//FloorStats 23
IF 
FB_BACnet_DAIKIN_MasterStation_III_No_6.StartStopStatus_064.bPresVal AND
FB_BACnet_DAIKIN_MasterStation_III_No_6.StartStopStatus_065.bPresVal AND
FB_BACnet_DAIKIN_MasterStation_III_No_6.StartStopStatus_066.bPresVal AND
FB_BACnet_DAIKIN_MasterStation_III_No_6.StartStopStatus_067.bPresVal AND
FB_BACnet_DAIKIN_MasterStation_III_No_6.StartStopStatus_068.bPresVal AND
FB_BACnet_DAIKIN_MasterStation_III_No_6.StartStopStatus_069.bPresVal AND
FB_BACnet_DAIKIN_MasterStation_III_No_6.StartStopStatus_070.bPresVal AND
FB_BACnet_DAIKIN_MasterStation_III_No_6.StartStopStatus_071.bPresVal AND
FB_BACnet_DAIKIN_MasterStation_III_No_6.StartStopStatus_072.bPresVal AND
FB_BACnet_DAIKIN_MasterStation_III_No_6.StartStopStatus_073.bPresVal AND
FB_BACnet_DAIKIN_MasterStation_III_No_6.StartStopStatus_074.bPresVal AND
FB_BACnet_DAIKIN_MasterStation_III_No_6.StartStopStatus_075.bPresVal AND
FB_BACnet_DAIKIN_MasterStation_III_No_6.StartStopStatus_076.bPresVal AND
FB_BACnet_DAIKIN_MasterStation_III_No_6.StartStopStatus_077.bPresVal AND
FB_BACnet_DAIKIN_MasterStation_III_No_6.StartStopStatus_078.bPresVal AND
FB_BACnet_DAIKIN_MasterStation_III_No_6.StartStopStatus_079.bPresVal AND
FB_BACnet_DAIKIN_MasterStation_III_No_6.StartStopStatus_080.bPresVal AND
FB_BACnet_DAIKIN_MasterStation_III_No_6.StartStopStatus_081.bPresVal AND
FB_BACnet_DAIKIN_MasterStation_III_No_6.StartStopStatus_082.bPresVal AND
FB_BACnet_DAIKIN_MasterStation_III_No_6.StartStopStatus_083.bPresVal AND
FB_BACnet_DAIKIN_MasterStation_III_No_6.StartStopStatus_224.bPresVal
THEN
	nFloorStatus23 := 1;
ELSIF
NOT FB_BACnet_DAIKIN_MasterStation_III_No_6.StartStopStatus_064.bPresVal AND
NOT FB_BACnet_DAIKIN_MasterStation_III_No_6.StartStopStatus_065.bPresVal AND
NOT FB_BACnet_DAIKIN_MasterStation_III_No_6.StartStopStatus_066.bPresVal AND
NOT FB_BACnet_DAIKIN_MasterStation_III_No_6.StartStopStatus_067.bPresVal AND
NOT FB_BACnet_DAIKIN_MasterStation_III_No_6.StartStopStatus_068.bPresVal AND
NOT FB_BACnet_DAIKIN_MasterStation_III_No_6.StartStopStatus_069.bPresVal AND
NOT FB_BACnet_DAIKIN_MasterStation_III_No_6.StartStopStatus_070.bPresVal AND
NOT FB_BACnet_DAIKIN_MasterStation_III_No_6.StartStopStatus_071.bPresVal AND
NOT FB_BACnet_DAIKIN_MasterStation_III_No_6.StartStopStatus_072.bPresVal AND
NOT FB_BACnet_DAIKIN_MasterStation_III_No_6.StartStopStatus_073.bPresVal AND
NOT FB_BACnet_DAIKIN_MasterStation_III_No_6.StartStopStatus_074.bPresVal AND
NOT FB_BACnet_DAIKIN_MasterStation_III_No_6.StartStopStatus_075.bPresVal AND
NOT FB_BACnet_DAIKIN_MasterStation_III_No_6.StartStopStatus_076.bPresVal AND
NOT FB_BACnet_DAIKIN_MasterStation_III_No_6.StartStopStatus_077.bPresVal AND
NOT FB_BACnet_DAIKIN_MasterStation_III_No_6.StartStopStatus_078.bPresVal AND
NOT FB_BACnet_DAIKIN_MasterStation_III_No_6.StartStopStatus_079.bPresVal AND
NOT FB_BACnet_DAIKIN_MasterStation_III_No_6.StartStopStatus_080.bPresVal AND
NOT FB_BACnet_DAIKIN_MasterStation_III_No_6.StartStopStatus_081.bPresVal AND
NOT FB_BACnet_DAIKIN_MasterStation_III_No_6.StartStopStatus_082.bPresVal AND
NOT FB_BACnet_DAIKIN_MasterStation_III_No_6.StartStopStatus_083.bPresVal AND
NOT FB_BACnet_DAIKIN_MasterStation_III_No_6.StartStopStatus_224.bPresVal
THEN
	nFloorStatus23 := 0;
ELSE
	nFloorStatus23 := 2;
END_IF

//FloorStats 25
IF 
FB_BACnet_DAIKIN_MasterStation_III_No_6.StartStopStatus_128.bPresVal AND
FB_BACnet_DAIKIN_MasterStation_III_No_6.StartStopStatus_129.bPresVal AND
FB_BACnet_DAIKIN_MasterStation_III_No_6.StartStopStatus_130.bPresVal AND
FB_BACnet_DAIKIN_MasterStation_III_No_6.StartStopStatus_131.bPresVal AND
FB_BACnet_DAIKIN_MasterStation_III_No_6.StartStopStatus_132.bPresVal AND
FB_BACnet_DAIKIN_MasterStation_III_No_6.StartStopStatus_133.bPresVal AND
//FB_BACnet_DAIKIN_MasterStation_III_No_6.StartStopStatus_134.bPresVal AND
//FB_BACnet_DAIKIN_MasterStation_III_No_6.StartStopStatus_135.bPresVal AND
FB_BACnet_DAIKIN_MasterStation_III_No_6.StartStopStatus_136.bPresVal AND
FB_BACnet_DAIKIN_MasterStation_III_No_6.StartStopStatus_137.bPresVal AND
FB_BACnet_DAIKIN_MasterStation_III_No_6.StartStopStatus_138.bPresVal AND
FB_BACnet_DAIKIN_MasterStation_III_No_6.StartStopStatus_139.bPresVal AND
FB_BACnet_DAIKIN_MasterStation_III_No_6.StartStopStatus_140.bPresVal AND
FB_BACnet_DAIKIN_MasterStation_III_No_6.StartStopStatus_141.bPresVal AND
FB_BACnet_DAIKIN_MasterStation_III_No_6.StartStopStatus_142.bPresVal AND
FB_BACnet_DAIKIN_MasterStation_III_No_6.StartStopStatus_143.bPresVal AND
FB_BACnet_DAIKIN_MasterStation_III_No_6.StartStopStatus_144.bPresVal AND
FB_BACnet_DAIKIN_MasterStation_III_No_6.StartStopStatus_145.bPresVal AND
FB_BACnet_DAIKIN_MasterStation_III_No_6.StartStopStatus_146.bPresVal AND
FB_BACnet_DAIKIN_MasterStation_III_No_6.StartStopStatus_147.bPresVal AND
FB_BACnet_DAIKIN_MasterStation_III_No_6.StartStopStatus_225.bPresVal AND
FB_BACnet_DAIKIN_MasterStation_III_No_6.StartStopStatus_241.bPresVal AND
FB_BACnet_DAIKIN_MasterStation_III_No_6.StartStopStatus_176.bPresVal
THEN
	nFloorStatus25 := 1;
ELSIF
NOT FB_BACnet_DAIKIN_MasterStation_III_No_6.StartStopStatus_128.bPresVal AND
NOT FB_BACnet_DAIKIN_MasterStation_III_No_6.StartStopStatus_129.bPresVal AND
NOT FB_BACnet_DAIKIN_MasterStation_III_No_6.StartStopStatus_130.bPresVal AND
NOT FB_BACnet_DAIKIN_MasterStation_III_No_6.StartStopStatus_131.bPresVal AND
NOT FB_BACnet_DAIKIN_MasterStation_III_No_6.StartStopStatus_132.bPresVal AND
NOT FB_BACnet_DAIKIN_MasterStation_III_No_6.StartStopStatus_133.bPresVal AND
//NOT FB_BACnet_DAIKIN_MasterStation_III_No_6.StartStopStatus_134.bPresVal AND
//NOT FB_BACnet_DAIKIN_MasterStation_III_No_6.StartStopStatus_135.bPresVal AND
NOT FB_BACnet_DAIKIN_MasterStation_III_No_6.StartStopStatus_136.bPresVal AND
NOT FB_BACnet_DAIKIN_MasterStation_III_No_6.StartStopStatus_137.bPresVal AND
NOT FB_BACnet_DAIKIN_MasterStation_III_No_6.StartStopStatus_138.bPresVal AND
NOT FB_BACnet_DAIKIN_MasterStation_III_No_6.StartStopStatus_139.bPresVal AND
NOT FB_BACnet_DAIKIN_MasterStation_III_No_6.StartStopStatus_140.bPresVal AND
NOT FB_BACnet_DAIKIN_MasterStation_III_No_6.StartStopStatus_141.bPresVal AND
NOT FB_BACnet_DAIKIN_MasterStation_III_No_6.StartStopStatus_142.bPresVal AND
NOT FB_BACnet_DAIKIN_MasterStation_III_No_6.StartStopStatus_143.bPresVal AND
NOT FB_BACnet_DAIKIN_MasterStation_III_No_6.StartStopStatus_144.bPresVal AND
NOT FB_BACnet_DAIKIN_MasterStation_III_No_6.StartStopStatus_145.bPresVal AND
NOT FB_BACnet_DAIKIN_MasterStation_III_No_6.StartStopStatus_146.bPresVal AND
NOT FB_BACnet_DAIKIN_MasterStation_III_No_6.StartStopStatus_147.bPresVal AND
NOT FB_BACnet_DAIKIN_MasterStation_III_No_6.StartStopStatus_225.bPresVal AND
NOT FB_BACnet_DAIKIN_MasterStation_III_No_6.StartStopStatus_241.bPresVal AND
NOT FB_BACnet_DAIKIN_MasterStation_III_No_6.StartStopStatus_176.bPresVal
THEN
	nFloorStatus25 := 0;
ELSE
	nFloorStatus25 := 2;
END_IF

//FloorStats 26
IF 
FB_BACnet_DAIKIN_MasterStation_III_No_6.StartStopStatus_192.bPresVal AND
FB_BACnet_DAIKIN_MasterStation_III_No_6.StartStopStatus_193.bPresVal AND
FB_BACnet_DAIKIN_MasterStation_III_No_6.StartStopStatus_194.bPresVal AND
FB_BACnet_DAIKIN_MasterStation_III_No_6.StartStopStatus_195.bPresVal AND
FB_BACnet_DAIKIN_MasterStation_III_No_6.StartStopStatus_196.bPresVal AND
FB_BACnet_DAIKIN_MasterStation_III_No_6.StartStopStatus_197.bPresVal AND
FB_BACnet_DAIKIN_MasterStation_III_No_6.StartStopStatus_198.bPresVal AND
FB_BACnet_DAIKIN_MasterStation_III_No_6.StartStopStatus_199.bPresVal AND
FB_BACnet_DAIKIN_MasterStation_III_No_6.StartStopStatus_200.bPresVal AND
FB_BACnet_DAIKIN_MasterStation_III_No_6.StartStopStatus_201.bPresVal AND
FB_BACnet_DAIKIN_MasterStation_III_No_6.StartStopStatus_202.bPresVal AND
FB_BACnet_DAIKIN_MasterStation_III_No_6.StartStopStatus_203.bPresVal AND
FB_BACnet_DAIKIN_MasterStation_III_No_6.StartStopStatus_204.bPresVal AND
FB_BACnet_DAIKIN_MasterStation_III_No_6.StartStopStatus_205.bPresVal AND
FB_BACnet_DAIKIN_MasterStation_III_No_6.StartStopStatus_206.bPresVal AND
FB_BACnet_DAIKIN_MasterStation_III_No_6.StartStopStatus_207.bPresVal AND
FB_BACnet_DAIKIN_MasterStation_III_No_6.StartStopStatus_208.bPresVal AND
FB_BACnet_DAIKIN_MasterStation_III_No_6.StartStopStatus_209.bPresVal AND
FB_BACnet_DAIKIN_MasterStation_III_No_6.StartStopStatus_210.bPresVal AND
FB_BACnet_DAIKIN_MasterStation_III_No_6.StartStopStatus_211.bPresVal AND
FB_BACnet_DAIKIN_MasterStation_III_No_6.StartStopStatus_226.bPresVal
THEN
	nFloorStatus26 := 1;
ELSIF
NOT FB_BACnet_DAIKIN_MasterStation_III_No_6.StartStopStatus_192.bPresVal AND
NOT FB_BACnet_DAIKIN_MasterStation_III_No_6.StartStopStatus_193.bPresVal AND
NOT FB_BACnet_DAIKIN_MasterStation_III_No_6.StartStopStatus_194.bPresVal AND
NOT FB_BACnet_DAIKIN_MasterStation_III_No_6.StartStopStatus_195.bPresVal AND
NOT FB_BACnet_DAIKIN_MasterStation_III_No_6.StartStopStatus_196.bPresVal AND
NOT FB_BACnet_DAIKIN_MasterStation_III_No_6.StartStopStatus_197.bPresVal AND
NOT FB_BACnet_DAIKIN_MasterStation_III_No_6.StartStopStatus_198.bPresVal AND
NOT FB_BACnet_DAIKIN_MasterStation_III_No_6.StartStopStatus_199.bPresVal AND
NOT FB_BACnet_DAIKIN_MasterStation_III_No_6.StartStopStatus_200.bPresVal AND
NOT FB_BACnet_DAIKIN_MasterStation_III_No_6.StartStopStatus_201.bPresVal AND
NOT FB_BACnet_DAIKIN_MasterStation_III_No_6.StartStopStatus_202.bPresVal AND
NOT FB_BACnet_DAIKIN_MasterStation_III_No_6.StartStopStatus_203.bPresVal AND
NOT FB_BACnet_DAIKIN_MasterStation_III_No_6.StartStopStatus_204.bPresVal AND
NOT FB_BACnet_DAIKIN_MasterStation_III_No_6.StartStopStatus_205.bPresVal AND
NOT FB_BACnet_DAIKIN_MasterStation_III_No_6.StartStopStatus_206.bPresVal AND
NOT FB_BACnet_DAIKIN_MasterStation_III_No_6.StartStopStatus_207.bPresVal AND
NOT FB_BACnet_DAIKIN_MasterStation_III_No_6.StartStopStatus_208.bPresVal AND
NOT FB_BACnet_DAIKIN_MasterStation_III_No_6.StartStopStatus_209.bPresVal AND
NOT FB_BACnet_DAIKIN_MasterStation_III_No_6.StartStopStatus_210.bPresVal AND
NOT FB_BACnet_DAIKIN_MasterStation_III_No_6.StartStopStatus_211.bPresVal AND
NOT FB_BACnet_DAIKIN_MasterStation_III_No_6.StartStopStatus_226.bPresVal
THEN
	nFloorStatus26 := 0;
ELSE
	nFloorStatus26 := 2;
END_IF

//FloorStats 27
IF 
FB_BACnet_DAIKIN_MasterStation_III_No_7.StartStopStatus_000.bPresVal AND
FB_BACnet_DAIKIN_MasterStation_III_No_7.StartStopStatus_001.bPresVal AND
FB_BACnet_DAIKIN_MasterStation_III_No_7.StartStopStatus_002.bPresVal AND
FB_BACnet_DAIKIN_MasterStation_III_No_7.StartStopStatus_003.bPresVal AND
FB_BACnet_DAIKIN_MasterStation_III_No_7.StartStopStatus_004.bPresVal AND
FB_BACnet_DAIKIN_MasterStation_III_No_7.StartStopStatus_005.bPresVal AND
FB_BACnet_DAIKIN_MasterStation_III_No_7.StartStopStatus_006.bPresVal AND
//FB_BACnet_DAIKIN_MasterStation_III_No_7.StartStopStatus_007.bPresVal AND
FB_BACnet_DAIKIN_MasterStation_III_No_7.StartStopStatus_008.bPresVal AND
//FB_BACnet_DAIKIN_MasterStation_III_No_7.StartStopStatus_009.bPresVal AND
FB_BACnet_DAIKIN_MasterStation_III_No_7.StartStopStatus_010.bPresVal AND
FB_BACnet_DAIKIN_MasterStation_III_No_7.StartStopStatus_011.bPresVal AND
FB_BACnet_DAIKIN_MasterStation_III_No_7.StartStopStatus_012.bPresVal AND
FB_BACnet_DAIKIN_MasterStation_III_No_7.StartStopStatus_013.bPresVal AND
FB_BACnet_DAIKIN_MasterStation_III_No_7.StartStopStatus_014.bPresVal AND
FB_BACnet_DAIKIN_MasterStation_III_No_7.StartStopStatus_015.bPresVal AND
FB_BACnet_DAIKIN_MasterStation_III_No_7.StartStopStatus_016.bPresVal AND
FB_BACnet_DAIKIN_MasterStation_III_No_7.StartStopStatus_017.bPresVal AND
FB_BACnet_DAIKIN_MasterStation_III_No_7.StartStopStatus_018.bPresVal AND
FB_BACnet_DAIKIN_MasterStation_III_No_7.StartStopStatus_019.bPresVal AND
FB_BACnet_DAIKIN_MasterStation_III_No_7.StartStopStatus_224.bPresVal
THEN
	nFloorStatus27 := 1;
ELSIF
NOT FB_BACnet_DAIKIN_MasterStation_III_No_7.StartStopStatus_000.bPresVal AND
NOT FB_BACnet_DAIKIN_MasterStation_III_No_7.StartStopStatus_001.bPresVal AND
NOT FB_BACnet_DAIKIN_MasterStation_III_No_7.StartStopStatus_002.bPresVal AND
NOT FB_BACnet_DAIKIN_MasterStation_III_No_7.StartStopStatus_003.bPresVal AND
NOT FB_BACnet_DAIKIN_MasterStation_III_No_7.StartStopStatus_004.bPresVal AND
NOT FB_BACnet_DAIKIN_MasterStation_III_No_7.StartStopStatus_005.bPresVal AND
NOT FB_BACnet_DAIKIN_MasterStation_III_No_7.StartStopStatus_006.bPresVal AND
//NOT FB_BACnet_DAIKIN_MasterStation_III_No_7.StartStopStatus_007.bPresVal AND
NOT FB_BACnet_DAIKIN_MasterStation_III_No_7.StartStopStatus_008.bPresVal AND
//NOT FB_BACnet_DAIKIN_MasterStation_III_No_7.StartStopStatus_009.bPresVal AND
NOT FB_BACnet_DAIKIN_MasterStation_III_No_7.StartStopStatus_010.bPresVal AND
NOT FB_BACnet_DAIKIN_MasterStation_III_No_7.StartStopStatus_011.bPresVal AND
NOT FB_BACnet_DAIKIN_MasterStation_III_No_7.StartStopStatus_012.bPresVal AND
NOT FB_BACnet_DAIKIN_MasterStation_III_No_7.StartStopStatus_013.bPresVal AND
NOT FB_BACnet_DAIKIN_MasterStation_III_No_7.StartStopStatus_014.bPresVal AND
NOT FB_BACnet_DAIKIN_MasterStation_III_No_7.StartStopStatus_015.bPresVal AND
NOT FB_BACnet_DAIKIN_MasterStation_III_No_7.StartStopStatus_016.bPresVal AND
NOT FB_BACnet_DAIKIN_MasterStation_III_No_7.StartStopStatus_017.bPresVal AND
NOT FB_BACnet_DAIKIN_MasterStation_III_No_7.StartStopStatus_018.bPresVal AND
NOT FB_BACnet_DAIKIN_MasterStation_III_No_7.StartStopStatus_019.bPresVal AND
NOT FB_BACnet_DAIKIN_MasterStation_III_No_7.StartStopStatus_224.bPresVal
THEN
	nFloorStatus27 := 0;
ELSE
	nFloorStatus27 := 2;
END_IF

//FloorStats 28
IF 
FB_BACnet_DAIKIN_MasterStation_III_No_7.StartStopStatus_064.bPresVal AND
FB_BACnet_DAIKIN_MasterStation_III_No_7.StartStopStatus_065.bPresVal AND
FB_BACnet_DAIKIN_MasterStation_III_No_7.StartStopStatus_066.bPresVal AND
FB_BACnet_DAIKIN_MasterStation_III_No_7.StartStopStatus_067.bPresVal AND
FB_BACnet_DAIKIN_MasterStation_III_No_7.StartStopStatus_068.bPresVal AND
FB_BACnet_DAIKIN_MasterStation_III_No_7.StartStopStatus_069.bPresVal AND
FB_BACnet_DAIKIN_MasterStation_III_No_7.StartStopStatus_070.bPresVal AND
FB_BACnet_DAIKIN_MasterStation_III_No_7.StartStopStatus_071.bPresVal AND
FB_BACnet_DAIKIN_MasterStation_III_No_7.StartStopStatus_072.bPresVal AND
FB_BACnet_DAIKIN_MasterStation_III_No_7.StartStopStatus_073.bPresVal AND
FB_BACnet_DAIKIN_MasterStation_III_No_7.StartStopStatus_074.bPresVal AND
FB_BACnet_DAIKIN_MasterStation_III_No_7.StartStopStatus_075.bPresVal AND
FB_BACnet_DAIKIN_MasterStation_III_No_7.StartStopStatus_076.bPresVal AND
FB_BACnet_DAIKIN_MasterStation_III_No_7.StartStopStatus_077.bPresVal AND
FB_BACnet_DAIKIN_MasterStation_III_No_7.StartStopStatus_078.bPresVal AND
FB_BACnet_DAIKIN_MasterStation_III_No_7.StartStopStatus_079.bPresVal AND
FB_BACnet_DAIKIN_MasterStation_III_No_7.StartStopStatus_080.bPresVal AND
FB_BACnet_DAIKIN_MasterStation_III_No_7.StartStopStatus_081.bPresVal AND
FB_BACnet_DAIKIN_MasterStation_III_No_7.StartStopStatus_082.bPresVal AND
FB_BACnet_DAIKIN_MasterStation_III_No_7.StartStopStatus_083.bPresVal AND
FB_BACnet_DAIKIN_MasterStation_III_No_7.StartStopStatus_225.bPresVal AND
FB_BACnet_DAIKIN_MasterStation_III_No_7.StartStopStatus_241.bPresVal AND
FB_BACnet_DAIKIN_MasterStation_III_No_7.StartStopStatus_112.bPresVal
THEN
	nFloorStatus28 := 1;
ELSIF
NOT FB_BACnet_DAIKIN_MasterStation_III_No_7.StartStopStatus_064.bPresVal AND
NOT FB_BACnet_DAIKIN_MasterStation_III_No_7.StartStopStatus_065.bPresVal AND
NOT FB_BACnet_DAIKIN_MasterStation_III_No_7.StartStopStatus_066.bPresVal AND
NOT FB_BACnet_DAIKIN_MasterStation_III_No_7.StartStopStatus_067.bPresVal AND
NOT FB_BACnet_DAIKIN_MasterStation_III_No_7.StartStopStatus_068.bPresVal AND
NOT FB_BACnet_DAIKIN_MasterStation_III_No_7.StartStopStatus_069.bPresVal AND
NOT FB_BACnet_DAIKIN_MasterStation_III_No_7.StartStopStatus_070.bPresVal AND
NOT FB_BACnet_DAIKIN_MasterStation_III_No_7.StartStopStatus_071.bPresVal AND
NOT FB_BACnet_DAIKIN_MasterStation_III_No_7.StartStopStatus_072.bPresVal AND
NOT FB_BACnet_DAIKIN_MasterStation_III_No_7.StartStopStatus_073.bPresVal AND
NOT FB_BACnet_DAIKIN_MasterStation_III_No_7.StartStopStatus_074.bPresVal AND
NOT FB_BACnet_DAIKIN_MasterStation_III_No_7.StartStopStatus_075.bPresVal AND
NOT FB_BACnet_DAIKIN_MasterStation_III_No_7.StartStopStatus_076.bPresVal AND
NOT FB_BACnet_DAIKIN_MasterStation_III_No_7.StartStopStatus_077.bPresVal AND
NOT FB_BACnet_DAIKIN_MasterStation_III_No_7.StartStopStatus_078.bPresVal AND
NOT FB_BACnet_DAIKIN_MasterStation_III_No_7.StartStopStatus_079.bPresVal AND
NOT FB_BACnet_DAIKIN_MasterStation_III_No_7.StartStopStatus_080.bPresVal AND
NOT FB_BACnet_DAIKIN_MasterStation_III_No_7.StartStopStatus_081.bPresVal AND
NOT FB_BACnet_DAIKIN_MasterStation_III_No_7.StartStopStatus_082.bPresVal AND
NOT FB_BACnet_DAIKIN_MasterStation_III_No_7.StartStopStatus_083.bPresVal AND
NOT FB_BACnet_DAIKIN_MasterStation_III_No_7.StartStopStatus_225.bPresVal AND
NOT FB_BACnet_DAIKIN_MasterStation_III_No_7.StartStopStatus_241.bPresVal AND
NOT FB_BACnet_DAIKIN_MasterStation_III_No_7.StartStopStatus_112.bPresVal
THEN
	nFloorStatus28 := 0;
ELSE
	nFloorStatus28 := 2;
END_IF

//FloorStats 29
IF 
FB_BACnet_DAIKIN_MasterStation_III_No_7.StartStopStatus_128.bPresVal AND
FB_BACnet_DAIKIN_MasterStation_III_No_7.StartStopStatus_129.bPresVal AND
FB_BACnet_DAIKIN_MasterStation_III_No_7.StartStopStatus_130.bPresVal AND
FB_BACnet_DAIKIN_MasterStation_III_No_7.StartStopStatus_131.bPresVal AND
FB_BACnet_DAIKIN_MasterStation_III_No_7.StartStopStatus_132.bPresVal AND
FB_BACnet_DAIKIN_MasterStation_III_No_7.StartStopStatus_133.bPresVal AND
FB_BACnet_DAIKIN_MasterStation_III_No_7.StartStopStatus_134.bPresVal AND
FB_BACnet_DAIKIN_MasterStation_III_No_7.StartStopStatus_135.bPresVal AND
FB_BACnet_DAIKIN_MasterStation_III_No_7.StartStopStatus_136.bPresVal AND
FB_BACnet_DAIKIN_MasterStation_III_No_7.StartStopStatus_137.bPresVal AND
FB_BACnet_DAIKIN_MasterStation_III_No_7.StartStopStatus_138.bPresVal AND
FB_BACnet_DAIKIN_MasterStation_III_No_7.StartStopStatus_139.bPresVal AND
FB_BACnet_DAIKIN_MasterStation_III_No_7.StartStopStatus_140.bPresVal AND
FB_BACnet_DAIKIN_MasterStation_III_No_7.StartStopStatus_141.bPresVal AND
FB_BACnet_DAIKIN_MasterStation_III_No_7.StartStopStatus_142.bPresVal AND
FB_BACnet_DAIKIN_MasterStation_III_No_7.StartStopStatus_143.bPresVal AND
FB_BACnet_DAIKIN_MasterStation_III_No_7.StartStopStatus_144.bPresVal AND
FB_BACnet_DAIKIN_MasterStation_III_No_7.StartStopStatus_145.bPresVal AND
FB_BACnet_DAIKIN_MasterStation_III_No_7.StartStopStatus_146.bPresVal AND
FB_BACnet_DAIKIN_MasterStation_III_No_7.StartStopStatus_147.bPresVal AND
FB_BACnet_DAIKIN_MasterStation_III_No_7.StartStopStatus_226.bPresVal AND
FB_BACnet_DAIKIN_MasterStation_III_No_7.StartStopStatus_148.bPresVal AND
FB_BACnet_DAIKIN_MasterStation_III_No_7.StartStopStatus_149.bPresVal
THEN
	nFloorStatus29 := 1;
ELSIF
NOT FB_BACnet_DAIKIN_MasterStation_III_No_7.StartStopStatus_128.bPresVal AND
NOT FB_BACnet_DAIKIN_MasterStation_III_No_7.StartStopStatus_129.bPresVal AND
NOT FB_BACnet_DAIKIN_MasterStation_III_No_7.StartStopStatus_130.bPresVal AND
NOT FB_BACnet_DAIKIN_MasterStation_III_No_7.StartStopStatus_131.bPresVal AND
NOT FB_BACnet_DAIKIN_MasterStation_III_No_7.StartStopStatus_132.bPresVal AND
NOT FB_BACnet_DAIKIN_MasterStation_III_No_7.StartStopStatus_133.bPresVal AND
NOT FB_BACnet_DAIKIN_MasterStation_III_No_7.StartStopStatus_134.bPresVal AND
NOT FB_BACnet_DAIKIN_MasterStation_III_No_7.StartStopStatus_135.bPresVal AND
NOT FB_BACnet_DAIKIN_MasterStation_III_No_7.StartStopStatus_136.bPresVal AND
NOT FB_BACnet_DAIKIN_MasterStation_III_No_7.StartStopStatus_137.bPresVal AND
NOT FB_BACnet_DAIKIN_MasterStation_III_No_7.StartStopStatus_138.bPresVal AND
NOT FB_BACnet_DAIKIN_MasterStation_III_No_7.StartStopStatus_139.bPresVal AND
NOT FB_BACnet_DAIKIN_MasterStation_III_No_7.StartStopStatus_140.bPresVal AND
NOT FB_BACnet_DAIKIN_MasterStation_III_No_7.StartStopStatus_141.bPresVal AND
NOT FB_BACnet_DAIKIN_MasterStation_III_No_7.StartStopStatus_142.bPresVal AND
NOT FB_BACnet_DAIKIN_MasterStation_III_No_7.StartStopStatus_143.bPresVal AND
NOT FB_BACnet_DAIKIN_MasterStation_III_No_7.StartStopStatus_144.bPresVal AND
NOT FB_BACnet_DAIKIN_MasterStation_III_No_7.StartStopStatus_145.bPresVal AND
NOT FB_BACnet_DAIKIN_MasterStation_III_No_7.StartStopStatus_146.bPresVal AND
NOT FB_BACnet_DAIKIN_MasterStation_III_No_7.StartStopStatus_147.bPresVal AND
NOT FB_BACnet_DAIKIN_MasterStation_III_No_7.StartStopStatus_226.bPresVal AND
NOT FB_BACnet_DAIKIN_MasterStation_III_No_7.StartStopStatus_148.bPresVal AND
NOT FB_BACnet_DAIKIN_MasterStation_III_No_7.StartStopStatus_149.bPresVal
THEN
	nFloorStatus29 := 0;
ELSE
	nFloorStatus29 := 2;
END_IF

//FloorStats 30
IF 
FB_BACnet_DAIKIN_MasterStation_III_No_7.StartStopStatus_192.bPresVal AND
FB_BACnet_DAIKIN_MasterStation_III_No_7.StartStopStatus_193.bPresVal AND
FB_BACnet_DAIKIN_MasterStation_III_No_7.StartStopStatus_194.bPresVal AND
FB_BACnet_DAIKIN_MasterStation_III_No_7.StartStopStatus_195.bPresVal AND
FB_BACnet_DAIKIN_MasterStation_III_No_7.StartStopStatus_196.bPresVal AND
FB_BACnet_DAIKIN_MasterStation_III_No_7.StartStopStatus_197.bPresVal AND
FB_BACnet_DAIKIN_MasterStation_III_No_7.StartStopStatus_198.bPresVal AND
FB_BACnet_DAIKIN_MasterStation_III_No_7.StartStopStatus_199.bPresVal AND
FB_BACnet_DAIKIN_MasterStation_III_No_7.StartStopStatus_200.bPresVal AND
FB_BACnet_DAIKIN_MasterStation_III_No_7.StartStopStatus_201.bPresVal AND
FB_BACnet_DAIKIN_MasterStation_III_No_7.StartStopStatus_202.bPresVal AND
FB_BACnet_DAIKIN_MasterStation_III_No_7.StartStopStatus_203.bPresVal AND
FB_BACnet_DAIKIN_MasterStation_III_No_7.StartStopStatus_204.bPresVal AND
FB_BACnet_DAIKIN_MasterStation_III_No_7.StartStopStatus_205.bPresVal AND
FB_BACnet_DAIKIN_MasterStation_III_No_7.StartStopStatus_206.bPresVal AND
FB_BACnet_DAIKIN_MasterStation_III_No_7.StartStopStatus_207.bPresVal AND
FB_BACnet_DAIKIN_MasterStation_III_No_7.StartStopStatus_208.bPresVal AND
FB_BACnet_DAIKIN_MasterStation_III_No_7.StartStopStatus_209.bPresVal AND
FB_BACnet_DAIKIN_MasterStation_III_No_7.StartStopStatus_210.bPresVal AND
FB_BACnet_DAIKIN_MasterStation_III_No_7.StartStopStatus_211.bPresVal AND
FB_BACnet_DAIKIN_MasterStation_III_No_7.StartStopStatus_212.bPresVal AND
FB_BACnet_DAIKIN_MasterStation_III_No_7.StartStopStatus_227.bPresVal
THEN
	nFloorStatus30 := 1;
ELSIF
NOT FB_BACnet_DAIKIN_MasterStation_III_No_7.StartStopStatus_192.bPresVal AND
NOT FB_BACnet_DAIKIN_MasterStation_III_No_7.StartStopStatus_193.bPresVal AND
NOT FB_BACnet_DAIKIN_MasterStation_III_No_7.StartStopStatus_194.bPresVal AND
NOT FB_BACnet_DAIKIN_MasterStation_III_No_7.StartStopStatus_195.bPresVal AND
NOT FB_BACnet_DAIKIN_MasterStation_III_No_7.StartStopStatus_196.bPresVal AND
NOT FB_BACnet_DAIKIN_MasterStation_III_No_7.StartStopStatus_197.bPresVal AND
NOT FB_BACnet_DAIKIN_MasterStation_III_No_7.StartStopStatus_198.bPresVal AND
NOT FB_BACnet_DAIKIN_MasterStation_III_No_7.StartStopStatus_199.bPresVal AND
NOT FB_BACnet_DAIKIN_MasterStation_III_No_7.StartStopStatus_200.bPresVal AND
NOT FB_BACnet_DAIKIN_MasterStation_III_No_7.StartStopStatus_201.bPresVal AND
NOT FB_BACnet_DAIKIN_MasterStation_III_No_7.StartStopStatus_202.bPresVal AND
NOT FB_BACnet_DAIKIN_MasterStation_III_No_7.StartStopStatus_203.bPresVal AND
NOT FB_BACnet_DAIKIN_MasterStation_III_No_7.StartStopStatus_204.bPresVal AND
NOT FB_BACnet_DAIKIN_MasterStation_III_No_7.StartStopStatus_205.bPresVal AND
NOT FB_BACnet_DAIKIN_MasterStation_III_No_7.StartStopStatus_206.bPresVal AND
NOT FB_BACnet_DAIKIN_MasterStation_III_No_7.StartStopStatus_207.bPresVal AND
NOT FB_BACnet_DAIKIN_MasterStation_III_No_7.StartStopStatus_208.bPresVal AND
NOT FB_BACnet_DAIKIN_MasterStation_III_No_7.StartStopStatus_209.bPresVal AND
NOT FB_BACnet_DAIKIN_MasterStation_III_No_7.StartStopStatus_210.bPresVal AND
NOT FB_BACnet_DAIKIN_MasterStation_III_No_7.StartStopStatus_211.bPresVal AND
NOT FB_BACnet_DAIKIN_MasterStation_III_No_7.StartStopStatus_212.bPresVal AND
NOT FB_BACnet_DAIKIN_MasterStation_III_No_7.StartStopStatus_227.bPresVal
THEN
	nFloorStatus30 := 0;
ELSE
	nFloorStatus30 := 2;
END_IF

//FloorStats 31
IF 
FB_BACnet_DAIKIN_MasterStation_III_No_8.StartStopStatus_000.bPresVal AND
FB_BACnet_DAIKIN_MasterStation_III_No_8.StartStopStatus_001.bPresVal AND
FB_BACnet_DAIKIN_MasterStation_III_No_8.StartStopStatus_002.bPresVal AND
FB_BACnet_DAIKIN_MasterStation_III_No_8.StartStopStatus_003.bPresVal AND
FB_BACnet_DAIKIN_MasterStation_III_No_8.StartStopStatus_004.bPresVal AND
FB_BACnet_DAIKIN_MasterStation_III_No_8.StartStopStatus_005.bPresVal AND
FB_BACnet_DAIKIN_MasterStation_III_No_8.StartStopStatus_006.bPresVal AND
FB_BACnet_DAIKIN_MasterStation_III_No_8.StartStopStatus_007.bPresVal AND
FB_BACnet_DAIKIN_MasterStation_III_No_8.StartStopStatus_008.bPresVal AND
FB_BACnet_DAIKIN_MasterStation_III_No_8.StartStopStatus_009.bPresVal AND
FB_BACnet_DAIKIN_MasterStation_III_No_8.StartStopStatus_010.bPresVal AND
FB_BACnet_DAIKIN_MasterStation_III_No_8.StartStopStatus_011.bPresVal AND
FB_BACnet_DAIKIN_MasterStation_III_No_8.StartStopStatus_012.bPresVal AND
FB_BACnet_DAIKIN_MasterStation_III_No_8.StartStopStatus_013.bPresVal AND
FB_BACnet_DAIKIN_MasterStation_III_No_8.StartStopStatus_014.bPresVal AND
FB_BACnet_DAIKIN_MasterStation_III_No_8.StartStopStatus_015.bPresVal AND
FB_BACnet_DAIKIN_MasterStation_III_No_8.StartStopStatus_016.bPresVal AND
FB_BACnet_DAIKIN_MasterStation_III_No_8.StartStopStatus_017.bPresVal AND
FB_BACnet_DAIKIN_MasterStation_III_No_8.StartStopStatus_018.bPresVal AND
FB_BACnet_DAIKIN_MasterStation_III_No_8.StartStopStatus_019.bPresVal AND
FB_BACnet_DAIKIN_MasterStation_III_No_8.StartStopStatus_020.bPresVal AND
FB_BACnet_DAIKIN_MasterStation_III_No_8.StartStopStatus_224.bPresVal AND
FB_BACnet_DAIKIN_MasterStation_III_No_8.StartStopStatus_241.bPresVal 
//FB_BACnet_DAIKIN_MasterStation_III_No_8.StartStopStatus_048.bPresVal
THEN
	nFloorStatus31 := 1;
ELSIF
NOT FB_BACnet_DAIKIN_MasterStation_III_No_8.StartStopStatus_000.bPresVal AND
NOT FB_BACnet_DAIKIN_MasterStation_III_No_8.StartStopStatus_001.bPresVal AND
NOT FB_BACnet_DAIKIN_MasterStation_III_No_8.StartStopStatus_002.bPresVal AND
NOT FB_BACnet_DAIKIN_MasterStation_III_No_8.StartStopStatus_003.bPresVal AND
NOT FB_BACnet_DAIKIN_MasterStation_III_No_8.StartStopStatus_004.bPresVal AND
NOT FB_BACnet_DAIKIN_MasterStation_III_No_8.StartStopStatus_005.bPresVal AND
NOT FB_BACnet_DAIKIN_MasterStation_III_No_8.StartStopStatus_006.bPresVal AND
NOT FB_BACnet_DAIKIN_MasterStation_III_No_8.StartStopStatus_007.bPresVal AND
NOT FB_BACnet_DAIKIN_MasterStation_III_No_8.StartStopStatus_008.bPresVal AND
NOT FB_BACnet_DAIKIN_MasterStation_III_No_8.StartStopStatus_009.bPresVal AND
NOT FB_BACnet_DAIKIN_MasterStation_III_No_8.StartStopStatus_010.bPresVal AND
NOT FB_BACnet_DAIKIN_MasterStation_III_No_8.StartStopStatus_011.bPresVal AND
NOT FB_BACnet_DAIKIN_MasterStation_III_No_8.StartStopStatus_012.bPresVal AND
NOT FB_BACnet_DAIKIN_MasterStation_III_No_8.StartStopStatus_013.bPresVal AND
NOT FB_BACnet_DAIKIN_MasterStation_III_No_8.StartStopStatus_014.bPresVal AND
NOT FB_BACnet_DAIKIN_MasterStation_III_No_8.StartStopStatus_015.bPresVal AND
NOT FB_BACnet_DAIKIN_MasterStation_III_No_8.StartStopStatus_016.bPresVal AND
NOT FB_BACnet_DAIKIN_MasterStation_III_No_8.StartStopStatus_017.bPresVal AND
NOT FB_BACnet_DAIKIN_MasterStation_III_No_8.StartStopStatus_018.bPresVal AND
NOT FB_BACnet_DAIKIN_MasterStation_III_No_8.StartStopStatus_019.bPresVal AND
NOT FB_BACnet_DAIKIN_MasterStation_III_No_8.StartStopStatus_020.bPresVal AND
NOT FB_BACnet_DAIKIN_MasterStation_III_No_8.StartStopStatus_224.bPresVal AND
NOT FB_BACnet_DAIKIN_MasterStation_III_No_8.StartStopStatus_241.bPresVal
//NOT FB_BACnet_DAIKIN_MasterStation_III_No_8.StartStopStatus_048.bPresVal
THEN
	nFloorStatus31 := 0;
ELSE
	nFloorStatus31 := 2;
END_IF

//FloorStats 32
IF 
FB_BACnet_DAIKIN_MasterStation_III_No_8.StartStopStatus_064.bPresVal AND
FB_BACnet_DAIKIN_MasterStation_III_No_8.StartStopStatus_065.bPresVal AND
FB_BACnet_DAIKIN_MasterStation_III_No_8.StartStopStatus_066.bPresVal AND
FB_BACnet_DAIKIN_MasterStation_III_No_8.StartStopStatus_067.bPresVal AND
FB_BACnet_DAIKIN_MasterStation_III_No_8.StartStopStatus_068.bPresVal AND
FB_BACnet_DAIKIN_MasterStation_III_No_8.StartStopStatus_069.bPresVal AND
FB_BACnet_DAIKIN_MasterStation_III_No_8.StartStopStatus_070.bPresVal AND
FB_BACnet_DAIKIN_MasterStation_III_No_8.StartStopStatus_071.bPresVal AND
FB_BACnet_DAIKIN_MasterStation_III_No_8.StartStopStatus_072.bPresVal AND
FB_BACnet_DAIKIN_MasterStation_III_No_8.StartStopStatus_073.bPresVal AND
FB_BACnet_DAIKIN_MasterStation_III_No_8.StartStopStatus_074.bPresVal AND
FB_BACnet_DAIKIN_MasterStation_III_No_8.StartStopStatus_075.bPresVal AND
FB_BACnet_DAIKIN_MasterStation_III_No_8.StartStopStatus_076.bPresVal AND
FB_BACnet_DAIKIN_MasterStation_III_No_8.StartStopStatus_077.bPresVal AND
FB_BACnet_DAIKIN_MasterStation_III_No_8.StartStopStatus_078.bPresVal AND
FB_BACnet_DAIKIN_MasterStation_III_No_8.StartStopStatus_079.bPresVal AND
FB_BACnet_DAIKIN_MasterStation_III_No_8.StartStopStatus_080.bPresVal AND
FB_BACnet_DAIKIN_MasterStation_III_No_8.StartStopStatus_081.bPresVal AND
FB_BACnet_DAIKIN_MasterStation_III_No_8.StartStopStatus_082.bPresVal AND
FB_BACnet_DAIKIN_MasterStation_III_No_8.StartStopStatus_083.bPresVal AND
FB_BACnet_DAIKIN_MasterStation_III_No_8.StartStopStatus_084.bPresVal AND
FB_BACnet_DAIKIN_MasterStation_III_No_8.StartStopStatus_085.bPresVal AND
FB_BACnet_DAIKIN_MasterStation_III_No_8.StartStopStatus_225.bPresVal
THEN
	nFloorStatus32 := 1;
ELSIF
NOT FB_BACnet_DAIKIN_MasterStation_III_No_8.StartStopStatus_064.bPresVal AND
NOT FB_BACnet_DAIKIN_MasterStation_III_No_8.StartStopStatus_065.bPresVal AND
NOT FB_BACnet_DAIKIN_MasterStation_III_No_8.StartStopStatus_066.bPresVal AND
NOT FB_BACnet_DAIKIN_MasterStation_III_No_8.StartStopStatus_067.bPresVal AND
NOT FB_BACnet_DAIKIN_MasterStation_III_No_8.StartStopStatus_068.bPresVal AND
NOT FB_BACnet_DAIKIN_MasterStation_III_No_8.StartStopStatus_069.bPresVal AND
NOT FB_BACnet_DAIKIN_MasterStation_III_No_8.StartStopStatus_070.bPresVal AND
NOT FB_BACnet_DAIKIN_MasterStation_III_No_8.StartStopStatus_071.bPresVal AND
NOT FB_BACnet_DAIKIN_MasterStation_III_No_8.StartStopStatus_072.bPresVal AND
NOT FB_BACnet_DAIKIN_MasterStation_III_No_8.StartStopStatus_073.bPresVal AND
NOT FB_BACnet_DAIKIN_MasterStation_III_No_8.StartStopStatus_074.bPresVal AND
NOT FB_BACnet_DAIKIN_MasterStation_III_No_8.StartStopStatus_075.bPresVal AND
NOT FB_BACnet_DAIKIN_MasterStation_III_No_8.StartStopStatus_076.bPresVal AND
NOT FB_BACnet_DAIKIN_MasterStation_III_No_8.StartStopStatus_077.bPresVal AND
NOT FB_BACnet_DAIKIN_MasterStation_III_No_8.StartStopStatus_078.bPresVal AND
NOT FB_BACnet_DAIKIN_MasterStation_III_No_8.StartStopStatus_079.bPresVal AND
NOT FB_BACnet_DAIKIN_MasterStation_III_No_8.StartStopStatus_080.bPresVal AND
NOT FB_BACnet_DAIKIN_MasterStation_III_No_8.StartStopStatus_081.bPresVal AND
NOT FB_BACnet_DAIKIN_MasterStation_III_No_8.StartStopStatus_082.bPresVal AND
NOT FB_BACnet_DAIKIN_MasterStation_III_No_8.StartStopStatus_083.bPresVal AND
NOT FB_BACnet_DAIKIN_MasterStation_III_No_8.StartStopStatus_084.bPresVal AND
NOT FB_BACnet_DAIKIN_MasterStation_III_No_8.StartStopStatus_085.bPresVal AND
NOT FB_BACnet_DAIKIN_MasterStation_III_No_8.StartStopStatus_225.bPresVal
THEN
	nFloorStatus32 := 0;
ELSE
	nFloorStatus32 := 2;
END_IF

//FloorStats 33
IF 
FB_BACnet_DAIKIN_MasterStation_III_No_8.StartStopStatus_128.bPresVal AND
FB_BACnet_DAIKIN_MasterStation_III_No_8.StartStopStatus_129.bPresVal AND
FB_BACnet_DAIKIN_MasterStation_III_No_8.StartStopStatus_130.bPresVal AND
FB_BACnet_DAIKIN_MasterStation_III_No_8.StartStopStatus_131.bPresVal AND
FB_BACnet_DAIKIN_MasterStation_III_No_8.StartStopStatus_132.bPresVal AND
FB_BACnet_DAIKIN_MasterStation_III_No_8.StartStopStatus_133.bPresVal AND
FB_BACnet_DAIKIN_MasterStation_III_No_8.StartStopStatus_134.bPresVal AND
FB_BACnet_DAIKIN_MasterStation_III_No_8.StartStopStatus_135.bPresVal AND
FB_BACnet_DAIKIN_MasterStation_III_No_8.StartStopStatus_136.bPresVal AND
FB_BACnet_DAIKIN_MasterStation_III_No_8.StartStopStatus_137.bPresVal AND
FB_BACnet_DAIKIN_MasterStation_III_No_8.StartStopStatus_138.bPresVal AND
FB_BACnet_DAIKIN_MasterStation_III_No_8.StartStopStatus_139.bPresVal AND
FB_BACnet_DAIKIN_MasterStation_III_No_8.StartStopStatus_140.bPresVal AND
FB_BACnet_DAIKIN_MasterStation_III_No_8.StartStopStatus_141.bPresVal AND
FB_BACnet_DAIKIN_MasterStation_III_No_8.StartStopStatus_142.bPresVal AND
FB_BACnet_DAIKIN_MasterStation_III_No_8.StartStopStatus_143.bPresVal AND
FB_BACnet_DAIKIN_MasterStation_III_No_8.StartStopStatus_144.bPresVal AND
FB_BACnet_DAIKIN_MasterStation_III_No_8.StartStopStatus_145.bPresVal AND
FB_BACnet_DAIKIN_MasterStation_III_No_8.StartStopStatus_146.bPresVal AND
FB_BACnet_DAIKIN_MasterStation_III_No_8.StartStopStatus_147.bPresVal AND
FB_BACnet_DAIKIN_MasterStation_III_No_8.StartStopStatus_148.bPresVal AND
FB_BACnet_DAIKIN_MasterStation_III_No_8.StartStopStatus_149.bPresVal AND
FB_BACnet_DAIKIN_MasterStation_III_No_8.StartStopStatus_226.bPresVal
THEN
	nFloorStatus33 := 1;
ELSIF
NOT FB_BACnet_DAIKIN_MasterStation_III_No_8.StartStopStatus_128.bPresVal AND
NOT FB_BACnet_DAIKIN_MasterStation_III_No_8.StartStopStatus_129.bPresVal AND
NOT FB_BACnet_DAIKIN_MasterStation_III_No_8.StartStopStatus_130.bPresVal AND
NOT FB_BACnet_DAIKIN_MasterStation_III_No_8.StartStopStatus_131.bPresVal AND
NOT FB_BACnet_DAIKIN_MasterStation_III_No_8.StartStopStatus_132.bPresVal AND
NOT FB_BACnet_DAIKIN_MasterStation_III_No_8.StartStopStatus_133.bPresVal AND
NOT FB_BACnet_DAIKIN_MasterStation_III_No_8.StartStopStatus_134.bPresVal AND
NOT FB_BACnet_DAIKIN_MasterStation_III_No_8.StartStopStatus_135.bPresVal AND
NOT FB_BACnet_DAIKIN_MasterStation_III_No_8.StartStopStatus_136.bPresVal AND
NOT FB_BACnet_DAIKIN_MasterStation_III_No_8.StartStopStatus_137.bPresVal AND
NOT FB_BACnet_DAIKIN_MasterStation_III_No_8.StartStopStatus_138.bPresVal AND
NOT FB_BACnet_DAIKIN_MasterStation_III_No_8.StartStopStatus_139.bPresVal AND
NOT FB_BACnet_DAIKIN_MasterStation_III_No_8.StartStopStatus_140.bPresVal AND
NOT FB_BACnet_DAIKIN_MasterStation_III_No_8.StartStopStatus_141.bPresVal AND
NOT FB_BACnet_DAIKIN_MasterStation_III_No_8.StartStopStatus_142.bPresVal AND
NOT FB_BACnet_DAIKIN_MasterStation_III_No_8.StartStopStatus_143.bPresVal AND
NOT FB_BACnet_DAIKIN_MasterStation_III_No_8.StartStopStatus_144.bPresVal AND
NOT FB_BACnet_DAIKIN_MasterStation_III_No_8.StartStopStatus_145.bPresVal AND
NOT FB_BACnet_DAIKIN_MasterStation_III_No_8.StartStopStatus_146.bPresVal AND
NOT FB_BACnet_DAIKIN_MasterStation_III_No_8.StartStopStatus_147.bPresVal AND
NOT FB_BACnet_DAIKIN_MasterStation_III_No_8.StartStopStatus_148.bPresVal AND
NOT FB_BACnet_DAIKIN_MasterStation_III_No_8.StartStopStatus_149.bPresVal AND
NOT FB_BACnet_DAIKIN_MasterStation_III_No_8.StartStopStatus_226.bPresVal
THEN
	nFloorStatus33 := 0;
ELSE
	nFloorStatus33 := 2;
END_IF

//FloorStats 35
IF 
FB_BACnet_DAIKIN_MasterStation_III_No_8.StartStopStatus_192.bPresVal AND
FB_BACnet_DAIKIN_MasterStation_III_No_8.StartStopStatus_193.bPresVal AND
FB_BACnet_DAIKIN_MasterStation_III_No_8.StartStopStatus_194.bPresVal AND
FB_BACnet_DAIKIN_MasterStation_III_No_8.StartStopStatus_195.bPresVal AND
FB_BACnet_DAIKIN_MasterStation_III_No_8.StartStopStatus_196.bPresVal AND
FB_BACnet_DAIKIN_MasterStation_III_No_8.StartStopStatus_197.bPresVal AND
FB_BACnet_DAIKIN_MasterStation_III_No_8.StartStopStatus_198.bPresVal AND
FB_BACnet_DAIKIN_MasterStation_III_No_8.StartStopStatus_199.bPresVal AND
FB_BACnet_DAIKIN_MasterStation_III_No_8.StartStopStatus_200.bPresVal AND
FB_BACnet_DAIKIN_MasterStation_III_No_8.StartStopStatus_201.bPresVal AND
FB_BACnet_DAIKIN_MasterStation_III_No_8.StartStopStatus_202.bPresVal AND
FB_BACnet_DAIKIN_MasterStation_III_No_8.StartStopStatus_203.bPresVal AND
FB_BACnet_DAIKIN_MasterStation_III_No_8.StartStopStatus_204.bPresVal AND
FB_BACnet_DAIKIN_MasterStation_III_No_8.StartStopStatus_205.bPresVal AND
FB_BACnet_DAIKIN_MasterStation_III_No_8.StartStopStatus_206.bPresVal AND
FB_BACnet_DAIKIN_MasterStation_III_No_8.StartStopStatus_207.bPresVal AND
FB_BACnet_DAIKIN_MasterStation_III_No_8.StartStopStatus_208.bPresVal AND
FB_BACnet_DAIKIN_MasterStation_III_No_8.StartStopStatus_209.bPresVal AND
FB_BACnet_DAIKIN_MasterStation_III_No_8.StartStopStatus_210.bPresVal AND
FB_BACnet_DAIKIN_MasterStation_III_No_8.StartStopStatus_211.bPresVal AND
FB_BACnet_DAIKIN_MasterStation_III_No_8.StartStopStatus_212.bPresVal AND
FB_BACnet_DAIKIN_MasterStation_III_No_8.StartStopStatus_213.bPresVal AND
FB_BACnet_DAIKIN_MasterStation_III_No_8.StartStopStatus_227.bPresVal AND
FB_BACnet_DAIKIN_MasterStation_III_No_8.StartStopStatus_243.bPresVal
//FB_BACnet_DAIKIN_MasterStation_III_No_8.StartStopStatus_242.bPresVal
THEN
	nFloorStatus35 := 1;
ELSIF
NOT FB_BACnet_DAIKIN_MasterStation_III_No_8.StartStopStatus_192.bPresVal AND
NOT FB_BACnet_DAIKIN_MasterStation_III_No_8.StartStopStatus_193.bPresVal AND
NOT FB_BACnet_DAIKIN_MasterStation_III_No_8.StartStopStatus_194.bPresVal AND
NOT FB_BACnet_DAIKIN_MasterStation_III_No_8.StartStopStatus_195.bPresVal AND
NOT FB_BACnet_DAIKIN_MasterStation_III_No_8.StartStopStatus_196.bPresVal AND
NOT FB_BACnet_DAIKIN_MasterStation_III_No_8.StartStopStatus_197.bPresVal AND
NOT FB_BACnet_DAIKIN_MasterStation_III_No_8.StartStopStatus_198.bPresVal AND
NOT FB_BACnet_DAIKIN_MasterStation_III_No_8.StartStopStatus_199.bPresVal AND
NOT FB_BACnet_DAIKIN_MasterStation_III_No_8.StartStopStatus_200.bPresVal AND
NOT FB_BACnet_DAIKIN_MasterStation_III_No_8.StartStopStatus_201.bPresVal AND
NOT FB_BACnet_DAIKIN_MasterStation_III_No_8.StartStopStatus_202.bPresVal AND
NOT FB_BACnet_DAIKIN_MasterStation_III_No_8.StartStopStatus_203.bPresVal AND
NOT FB_BACnet_DAIKIN_MasterStation_III_No_8.StartStopStatus_204.bPresVal AND
NOT FB_BACnet_DAIKIN_MasterStation_III_No_8.StartStopStatus_205.bPresVal AND
NOT FB_BACnet_DAIKIN_MasterStation_III_No_8.StartStopStatus_206.bPresVal AND
NOT FB_BACnet_DAIKIN_MasterStation_III_No_8.StartStopStatus_207.bPresVal AND
NOT FB_BACnet_DAIKIN_MasterStation_III_No_8.StartStopStatus_208.bPresVal AND
NOT FB_BACnet_DAIKIN_MasterStation_III_No_8.StartStopStatus_209.bPresVal AND
NOT FB_BACnet_DAIKIN_MasterStation_III_No_8.StartStopStatus_210.bPresVal AND
NOT FB_BACnet_DAIKIN_MasterStation_III_No_8.StartStopStatus_211.bPresVal AND
NOT FB_BACnet_DAIKIN_MasterStation_III_No_8.StartStopStatus_212.bPresVal AND
NOT FB_BACnet_DAIKIN_MasterStation_III_No_8.StartStopStatus_213.bPresVal AND
NOT FB_BACnet_DAIKIN_MasterStation_III_No_8.StartStopStatus_227.bPresVal AND
NOT FB_BACnet_DAIKIN_MasterStation_III_No_8.StartStopStatus_243.bPresVal 
//NOT FB_BACnet_DAIKIN_MasterStation_III_No_8.StartStopStatus_242.bPresVal
THEN
	nFloorStatus35 := 0;
ELSE
	nFloorStatus35 := 2;
END_IF

//FloorStats 36
IF 
FB_BACnet_DAIKIN_MasterStation_III_No_9.StartStopStatus_000.bPresVal AND
FB_BACnet_DAIKIN_MasterStation_III_No_9.StartStopStatus_001.bPresVal AND
FB_BACnet_DAIKIN_MasterStation_III_No_9.StartStopStatus_002.bPresVal AND
FB_BACnet_DAIKIN_MasterStation_III_No_9.StartStopStatus_003.bPresVal AND
FB_BACnet_DAIKIN_MasterStation_III_No_9.StartStopStatus_004.bPresVal AND
FB_BACnet_DAIKIN_MasterStation_III_No_9.StartStopStatus_005.bPresVal AND
FB_BACnet_DAIKIN_MasterStation_III_No_9.StartStopStatus_006.bPresVal AND
FB_BACnet_DAIKIN_MasterStation_III_No_9.StartStopStatus_007.bPresVal AND
FB_BACnet_DAIKIN_MasterStation_III_No_9.StartStopStatus_008.bPresVal AND
FB_BACnet_DAIKIN_MasterStation_III_No_9.StartStopStatus_009.bPresVal AND
FB_BACnet_DAIKIN_MasterStation_III_No_9.StartStopStatus_010.bPresVal AND
FB_BACnet_DAIKIN_MasterStation_III_No_9.StartStopStatus_011.bPresVal AND
FB_BACnet_DAIKIN_MasterStation_III_No_9.StartStopStatus_012.bPresVal AND
FB_BACnet_DAIKIN_MasterStation_III_No_9.StartStopStatus_013.bPresVal AND
FB_BACnet_DAIKIN_MasterStation_III_No_9.StartStopStatus_014.bPresVal AND
FB_BACnet_DAIKIN_MasterStation_III_No_9.StartStopStatus_015.bPresVal AND
FB_BACnet_DAIKIN_MasterStation_III_No_9.StartStopStatus_016.bPresVal AND
FB_BACnet_DAIKIN_MasterStation_III_No_9.StartStopStatus_017.bPresVal AND
FB_BACnet_DAIKIN_MasterStation_III_No_9.StartStopStatus_018.bPresVal AND
FB_BACnet_DAIKIN_MasterStation_III_No_9.StartStopStatus_019.bPresVal AND
FB_BACnet_DAIKIN_MasterStation_III_No_9.StartStopStatus_020.bPresVal AND
FB_BACnet_DAIKIN_MasterStation_III_No_9.StartStopStatus_021.bPresVal AND
FB_BACnet_DAIKIN_MasterStation_III_No_9.StartStopStatus_224.bPresVal
THEN
	nFloorStatus36 := 1;
ELSIF
NOT FB_BACnet_DAIKIN_MasterStation_III_No_9.StartStopStatus_000.bPresVal AND
NOT FB_BACnet_DAIKIN_MasterStation_III_No_9.StartStopStatus_001.bPresVal AND
NOT FB_BACnet_DAIKIN_MasterStation_III_No_9.StartStopStatus_002.bPresVal AND
NOT FB_BACnet_DAIKIN_MasterStation_III_No_9.StartStopStatus_003.bPresVal AND
NOT FB_BACnet_DAIKIN_MasterStation_III_No_9.StartStopStatus_004.bPresVal AND
NOT FB_BACnet_DAIKIN_MasterStation_III_No_9.StartStopStatus_005.bPresVal AND
NOT FB_BACnet_DAIKIN_MasterStation_III_No_9.StartStopStatus_006.bPresVal AND
NOT FB_BACnet_DAIKIN_MasterStation_III_No_9.StartStopStatus_007.bPresVal AND
NOT FB_BACnet_DAIKIN_MasterStation_III_No_9.StartStopStatus_008.bPresVal AND
NOT FB_BACnet_DAIKIN_MasterStation_III_No_9.StartStopStatus_009.bPresVal AND
NOT FB_BACnet_DAIKIN_MasterStation_III_No_9.StartStopStatus_010.bPresVal AND
NOT FB_BACnet_DAIKIN_MasterStation_III_No_9.StartStopStatus_011.bPresVal AND
NOT FB_BACnet_DAIKIN_MasterStation_III_No_9.StartStopStatus_012.bPresVal AND
NOT FB_BACnet_DAIKIN_MasterStation_III_No_9.StartStopStatus_013.bPresVal AND
NOT FB_BACnet_DAIKIN_MasterStation_III_No_9.StartStopStatus_014.bPresVal AND
NOT FB_BACnet_DAIKIN_MasterStation_III_No_9.StartStopStatus_015.bPresVal AND
NOT FB_BACnet_DAIKIN_MasterStation_III_No_9.StartStopStatus_016.bPresVal AND
NOT FB_BACnet_DAIKIN_MasterStation_III_No_9.StartStopStatus_017.bPresVal AND
NOT FB_BACnet_DAIKIN_MasterStation_III_No_9.StartStopStatus_018.bPresVal AND
NOT FB_BACnet_DAIKIN_MasterStation_III_No_9.StartStopStatus_019.bPresVal AND
NOT FB_BACnet_DAIKIN_MasterStation_III_No_9.StartStopStatus_020.bPresVal AND
NOT FB_BACnet_DAIKIN_MasterStation_III_No_9.StartStopStatus_021.bPresVal AND
NOT FB_BACnet_DAIKIN_MasterStation_III_No_9.StartStopStatus_224.bPresVal
THEN
	nFloorStatus36 := 0;
ELSE
	nFloorStatus36 := 2;
END_IF

//FloorStats 37
IF 
FB_BACnet_DAIKIN_MasterStation_III_No_9.StartStopStatus_064.bPresVal AND
FB_BACnet_DAIKIN_MasterStation_III_No_9.StartStopStatus_065.bPresVal AND
FB_BACnet_DAIKIN_MasterStation_III_No_9.StartStopStatus_066.bPresVal AND
FB_BACnet_DAIKIN_MasterStation_III_No_9.StartStopStatus_067.bPresVal AND
FB_BACnet_DAIKIN_MasterStation_III_No_9.StartStopStatus_068.bPresVal AND
FB_BACnet_DAIKIN_MasterStation_III_No_9.StartStopStatus_069.bPresVal AND
FB_BACnet_DAIKIN_MasterStation_III_No_9.StartStopStatus_070.bPresVal AND
FB_BACnet_DAIKIN_MasterStation_III_No_9.StartStopStatus_071.bPresVal AND
FB_BACnet_DAIKIN_MasterStation_III_No_9.StartStopStatus_072.bPresVal AND
FB_BACnet_DAIKIN_MasterStation_III_No_9.StartStopStatus_073.bPresVal AND
FB_BACnet_DAIKIN_MasterStation_III_No_9.StartStopStatus_074.bPresVal AND
FB_BACnet_DAIKIN_MasterStation_III_No_9.StartStopStatus_075.bPresVal AND
FB_BACnet_DAIKIN_MasterStation_III_No_9.StartStopStatus_076.bPresVal AND
FB_BACnet_DAIKIN_MasterStation_III_No_9.StartStopStatus_077.bPresVal AND
FB_BACnet_DAIKIN_MasterStation_III_No_9.StartStopStatus_078.bPresVal AND
FB_BACnet_DAIKIN_MasterStation_III_No_9.StartStopStatus_079.bPresVal AND
FB_BACnet_DAIKIN_MasterStation_III_No_9.StartStopStatus_080.bPresVal AND
FB_BACnet_DAIKIN_MasterStation_III_No_9.StartStopStatus_081.bPresVal AND
FB_BACnet_DAIKIN_MasterStation_III_No_9.StartStopStatus_082.bPresVal AND
FB_BACnet_DAIKIN_MasterStation_III_No_9.StartStopStatus_083.bPresVal AND
FB_BACnet_DAIKIN_MasterStation_III_No_9.StartStopStatus_084.bPresVal AND
FB_BACnet_DAIKIN_MasterStation_III_No_9.StartStopStatus_085.bPresVal AND
FB_BACnet_DAIKIN_MasterStation_III_No_9.StartStopStatus_225.bPresVal
THEN
	nFloorStatus37 := 1;
ELSIF
NOT FB_BACnet_DAIKIN_MasterStation_III_No_9.StartStopStatus_064.bPresVal AND
NOT FB_BACnet_DAIKIN_MasterStation_III_No_9.StartStopStatus_065.bPresVal AND
NOT FB_BACnet_DAIKIN_MasterStation_III_No_9.StartStopStatus_066.bPresVal AND
NOT FB_BACnet_DAIKIN_MasterStation_III_No_9.StartStopStatus_067.bPresVal AND
NOT FB_BACnet_DAIKIN_MasterStation_III_No_9.StartStopStatus_068.bPresVal AND
NOT FB_BACnet_DAIKIN_MasterStation_III_No_9.StartStopStatus_069.bPresVal AND
NOT FB_BACnet_DAIKIN_MasterStation_III_No_9.StartStopStatus_070.bPresVal AND
NOT FB_BACnet_DAIKIN_MasterStation_III_No_9.StartStopStatus_071.bPresVal AND
NOT FB_BACnet_DAIKIN_MasterStation_III_No_9.StartStopStatus_072.bPresVal AND
NOT FB_BACnet_DAIKIN_MasterStation_III_No_9.StartStopStatus_073.bPresVal AND
NOT FB_BACnet_DAIKIN_MasterStation_III_No_9.StartStopStatus_074.bPresVal AND
NOT FB_BACnet_DAIKIN_MasterStation_III_No_9.StartStopStatus_075.bPresVal AND
NOT FB_BACnet_DAIKIN_MasterStation_III_No_9.StartStopStatus_076.bPresVal AND
NOT FB_BACnet_DAIKIN_MasterStation_III_No_9.StartStopStatus_077.bPresVal AND
NOT FB_BACnet_DAIKIN_MasterStation_III_No_9.StartStopStatus_078.bPresVal AND
NOT FB_BACnet_DAIKIN_MasterStation_III_No_9.StartStopStatus_079.bPresVal AND
NOT FB_BACnet_DAIKIN_MasterStation_III_No_9.StartStopStatus_080.bPresVal AND
NOT FB_BACnet_DAIKIN_MasterStation_III_No_9.StartStopStatus_081.bPresVal AND
NOT FB_BACnet_DAIKIN_MasterStation_III_No_9.StartStopStatus_082.bPresVal AND
NOT FB_BACnet_DAIKIN_MasterStation_III_No_9.StartStopStatus_083.bPresVal AND
NOT FB_BACnet_DAIKIN_MasterStation_III_No_9.StartStopStatus_084.bPresVal AND
NOT FB_BACnet_DAIKIN_MasterStation_III_No_9.StartStopStatus_085.bPresVal AND
NOT FB_BACnet_DAIKIN_MasterStation_III_No_9.StartStopStatus_225.bPresVal
THEN
	nFloorStatus37 := 0;
ELSE
	nFloorStatus37 := 2;
END_IF

//FloorStats 38
IF 
FB_BACnet_DAIKIN_MasterStation_III_No_9.StartStopStatus_128.bPresVal AND
FB_BACnet_DAIKIN_MasterStation_III_No_9.StartStopStatus_129.bPresVal AND
FB_BACnet_DAIKIN_MasterStation_III_No_9.StartStopStatus_130.bPresVal AND
FB_BACnet_DAIKIN_MasterStation_III_No_9.StartStopStatus_131.bPresVal AND
FB_BACnet_DAIKIN_MasterStation_III_No_9.StartStopStatus_132.bPresVal AND
FB_BACnet_DAIKIN_MasterStation_III_No_9.StartStopStatus_133.bPresVal AND
FB_BACnet_DAIKIN_MasterStation_III_No_9.StartStopStatus_134.bPresVal AND
FB_BACnet_DAIKIN_MasterStation_III_No_9.StartStopStatus_135.bPresVal AND
FB_BACnet_DAIKIN_MasterStation_III_No_9.StartStopStatus_136.bPresVal AND
FB_BACnet_DAIKIN_MasterStation_III_No_9.StartStopStatus_137.bPresVal AND
FB_BACnet_DAIKIN_MasterStation_III_No_9.StartStopStatus_138.bPresVal AND
FB_BACnet_DAIKIN_MasterStation_III_No_9.StartStopStatus_139.bPresVal AND
FB_BACnet_DAIKIN_MasterStation_III_No_9.StartStopStatus_140.bPresVal AND
FB_BACnet_DAIKIN_MasterStation_III_No_9.StartStopStatus_141.bPresVal AND
FB_BACnet_DAIKIN_MasterStation_III_No_9.StartStopStatus_142.bPresVal AND
FB_BACnet_DAIKIN_MasterStation_III_No_9.StartStopStatus_143.bPresVal AND
FB_BACnet_DAIKIN_MasterStation_III_No_9.StartStopStatus_144.bPresVal AND
FB_BACnet_DAIKIN_MasterStation_III_No_9.StartStopStatus_145.bPresVal AND
FB_BACnet_DAIKIN_MasterStation_III_No_9.StartStopStatus_146.bPresVal AND
FB_BACnet_DAIKIN_MasterStation_III_No_9.StartStopStatus_147.bPresVal AND
FB_BACnet_DAIKIN_MasterStation_III_No_9.StartStopStatus_148.bPresVal AND
FB_BACnet_DAIKIN_MasterStation_III_No_9.StartStopStatus_149.bPresVal AND
FB_BACnet_DAIKIN_MasterStation_III_No_9.StartStopStatus_226.bPresVal AND
FB_BACnet_DAIKIN_MasterStation_III_No_9.StartStopStatus_241.bPresVal AND
FB_BACnet_DAIKIN_MasterStation_III_No_9.StartStopStatus_176.bPresVal
THEN
	nFloorStatus38 := 1;
ELSIF
NOT FB_BACnet_DAIKIN_MasterStation_III_No_9.StartStopStatus_128.bPresVal AND
NOT FB_BACnet_DAIKIN_MasterStation_III_No_9.StartStopStatus_129.bPresVal AND
NOT FB_BACnet_DAIKIN_MasterStation_III_No_9.StartStopStatus_130.bPresVal AND
NOT FB_BACnet_DAIKIN_MasterStation_III_No_9.StartStopStatus_131.bPresVal AND
NOT FB_BACnet_DAIKIN_MasterStation_III_No_9.StartStopStatus_132.bPresVal AND
NOT FB_BACnet_DAIKIN_MasterStation_III_No_9.StartStopStatus_133.bPresVal AND
NOT FB_BACnet_DAIKIN_MasterStation_III_No_9.StartStopStatus_134.bPresVal AND
NOT FB_BACnet_DAIKIN_MasterStation_III_No_9.StartStopStatus_135.bPresVal AND
NOT FB_BACnet_DAIKIN_MasterStation_III_No_9.StartStopStatus_136.bPresVal AND
NOT FB_BACnet_DAIKIN_MasterStation_III_No_9.StartStopStatus_137.bPresVal AND
NOT FB_BACnet_DAIKIN_MasterStation_III_No_9.StartStopStatus_138.bPresVal AND
NOT FB_BACnet_DAIKIN_MasterStation_III_No_9.StartStopStatus_139.bPresVal AND
NOT FB_BACnet_DAIKIN_MasterStation_III_No_9.StartStopStatus_140.bPresVal AND
NOT FB_BACnet_DAIKIN_MasterStation_III_No_9.StartStopStatus_141.bPresVal AND
NOT FB_BACnet_DAIKIN_MasterStation_III_No_9.StartStopStatus_142.bPresVal AND
NOT FB_BACnet_DAIKIN_MasterStation_III_No_9.StartStopStatus_143.bPresVal AND
NOT FB_BACnet_DAIKIN_MasterStation_III_No_9.StartStopStatus_144.bPresVal AND
NOT FB_BACnet_DAIKIN_MasterStation_III_No_9.StartStopStatus_145.bPresVal AND
NOT FB_BACnet_DAIKIN_MasterStation_III_No_9.StartStopStatus_146.bPresVal AND
NOT FB_BACnet_DAIKIN_MasterStation_III_No_9.StartStopStatus_147.bPresVal AND
NOT FB_BACnet_DAIKIN_MasterStation_III_No_9.StartStopStatus_148.bPresVal AND
NOT FB_BACnet_DAIKIN_MasterStation_III_No_9.StartStopStatus_149.bPresVal AND
NOT FB_BACnet_DAIKIN_MasterStation_III_No_9.StartStopStatus_226.bPresVal AND
NOT FB_BACnet_DAIKIN_MasterStation_III_No_9.StartStopStatus_241.bPresVal AND
NOT FB_BACnet_DAIKIN_MasterStation_III_No_9.StartStopStatus_176.bPresVal
THEN
	nFloorStatus38 := 0;
ELSE
	nFloorStatus38 := 2;
END_IF

//FloorStats 39
IF 
FB_BACnet_DAIKIN_MasterStation_III_No_9.StartStopStatus_192.bPresVal AND
FB_BACnet_DAIKIN_MasterStation_III_No_9.StartStopStatus_193.bPresVal AND
FB_BACnet_DAIKIN_MasterStation_III_No_9.StartStopStatus_194.bPresVal AND
FB_BACnet_DAIKIN_MasterStation_III_No_9.StartStopStatus_195.bPresVal AND
FB_BACnet_DAIKIN_MasterStation_III_No_9.StartStopStatus_196.bPresVal AND
FB_BACnet_DAIKIN_MasterStation_III_No_9.StartStopStatus_197.bPresVal AND
FB_BACnet_DAIKIN_MasterStation_III_No_9.StartStopStatus_198.bPresVal AND
FB_BACnet_DAIKIN_MasterStation_III_No_9.StartStopStatus_199.bPresVal AND
FB_BACnet_DAIKIN_MasterStation_III_No_9.StartStopStatus_200.bPresVal AND
FB_BACnet_DAIKIN_MasterStation_III_No_9.StartStopStatus_201.bPresVal AND
FB_BACnet_DAIKIN_MasterStation_III_No_9.StartStopStatus_202.bPresVal AND
FB_BACnet_DAIKIN_MasterStation_III_No_9.StartStopStatus_203.bPresVal AND
FB_BACnet_DAIKIN_MasterStation_III_No_9.StartStopStatus_204.bPresVal AND
FB_BACnet_DAIKIN_MasterStation_III_No_9.StartStopStatus_205.bPresVal AND
FB_BACnet_DAIKIN_MasterStation_III_No_9.StartStopStatus_206.bPresVal AND
FB_BACnet_DAIKIN_MasterStation_III_No_9.StartStopStatus_207.bPresVal AND
FB_BACnet_DAIKIN_MasterStation_III_No_9.StartStopStatus_208.bPresVal AND
FB_BACnet_DAIKIN_MasterStation_III_No_9.StartStopStatus_209.bPresVal AND
FB_BACnet_DAIKIN_MasterStation_III_No_9.StartStopStatus_210.bPresVal AND
FB_BACnet_DAIKIN_MasterStation_III_No_9.StartStopStatus_211.bPresVal AND
FB_BACnet_DAIKIN_MasterStation_III_No_9.StartStopStatus_212.bPresVal AND
FB_BACnet_DAIKIN_MasterStation_III_No_9.StartStopStatus_213.bPresVal AND
FB_BACnet_DAIKIN_MasterStation_III_No_9.StartStopStatus_227.bPresVal
THEN
	nFloorStatus39 := 1;
ELSIF
NOT FB_BACnet_DAIKIN_MasterStation_III_No_9.StartStopStatus_192.bPresVal AND
NOT FB_BACnet_DAIKIN_MasterStation_III_No_9.StartStopStatus_193.bPresVal AND
NOT FB_BACnet_DAIKIN_MasterStation_III_No_9.StartStopStatus_194.bPresVal AND
NOT FB_BACnet_DAIKIN_MasterStation_III_No_9.StartStopStatus_195.bPresVal AND
NOT FB_BACnet_DAIKIN_MasterStation_III_No_9.StartStopStatus_196.bPresVal AND
NOT FB_BACnet_DAIKIN_MasterStation_III_No_9.StartStopStatus_197.bPresVal AND
NOT FB_BACnet_DAIKIN_MasterStation_III_No_9.StartStopStatus_198.bPresVal AND
NOT FB_BACnet_DAIKIN_MasterStation_III_No_9.StartStopStatus_199.bPresVal AND
NOT FB_BACnet_DAIKIN_MasterStation_III_No_9.StartStopStatus_200.bPresVal AND
NOT FB_BACnet_DAIKIN_MasterStation_III_No_9.StartStopStatus_201.bPresVal AND
NOT FB_BACnet_DAIKIN_MasterStation_III_No_9.StartStopStatus_202.bPresVal AND
NOT FB_BACnet_DAIKIN_MasterStation_III_No_9.StartStopStatus_203.bPresVal AND
NOT FB_BACnet_DAIKIN_MasterStation_III_No_9.StartStopStatus_204.bPresVal AND
NOT FB_BACnet_DAIKIN_MasterStation_III_No_9.StartStopStatus_205.bPresVal AND
NOT FB_BACnet_DAIKIN_MasterStation_III_No_9.StartStopStatus_206.bPresVal AND
NOT FB_BACnet_DAIKIN_MasterStation_III_No_9.StartStopStatus_207.bPresVal AND
NOT FB_BACnet_DAIKIN_MasterStation_III_No_9.StartStopStatus_208.bPresVal AND
NOT FB_BACnet_DAIKIN_MasterStation_III_No_9.StartStopStatus_209.bPresVal AND
NOT FB_BACnet_DAIKIN_MasterStation_III_No_9.StartStopStatus_210.bPresVal AND
NOT FB_BACnet_DAIKIN_MasterStation_III_No_9.StartStopStatus_211.bPresVal AND
NOT FB_BACnet_DAIKIN_MasterStation_III_No_9.StartStopStatus_212.bPresVal AND
NOT FB_BACnet_DAIKIN_MasterStation_III_No_9.StartStopStatus_213.bPresVal AND
NOT FB_BACnet_DAIKIN_MasterStation_III_No_9.StartStopStatus_227.bPresVal
THEN
	nFloorStatus39 := 0;
ELSE
	nFloorStatus39 := 2;
END_IF

//FloorStats 50
IF 
FB_BACnet_DAIKIN_MasterStation_III_No_10.StartStopStatus_000.bPresVal AND
FB_BACnet_DAIKIN_MasterStation_III_No_10.StartStopStatus_001.bPresVal AND
FB_BACnet_DAIKIN_MasterStation_III_No_10.StartStopStatus_002.bPresVal AND
FB_BACnet_DAIKIN_MasterStation_III_No_10.StartStopStatus_003.bPresVal AND
FB_BACnet_DAIKIN_MasterStation_III_No_10.StartStopStatus_004.bPresVal AND
FB_BACnet_DAIKIN_MasterStation_III_No_10.StartStopStatus_005.bPresVal AND
FB_BACnet_DAIKIN_MasterStation_III_No_10.StartStopStatus_006.bPresVal AND
FB_BACnet_DAIKIN_MasterStation_III_No_10.StartStopStatus_007.bPresVal AND
FB_BACnet_DAIKIN_MasterStation_III_No_10.StartStopStatus_008.bPresVal AND
FB_BACnet_DAIKIN_MasterStation_III_No_10.StartStopStatus_009.bPresVal AND
FB_BACnet_DAIKIN_MasterStation_III_No_10.StartStopStatus_010.bPresVal AND
FB_BACnet_DAIKIN_MasterStation_III_No_10.StartStopStatus_011.bPresVal AND
FB_BACnet_DAIKIN_MasterStation_III_No_10.StartStopStatus_012.bPresVal AND
FB_BACnet_DAIKIN_MasterStation_III_No_10.StartStopStatus_013.bPresVal AND
FB_BACnet_DAIKIN_MasterStation_III_No_10.StartStopStatus_014.bPresVal AND
FB_BACnet_DAIKIN_MasterStation_III_No_10.StartStopStatus_015.bPresVal AND
FB_BACnet_DAIKIN_MasterStation_III_No_10.StartStopStatus_016.bPresVal AND
FB_BACnet_DAIKIN_MasterStation_III_No_10.StartStopStatus_017.bPresVal AND
FB_BACnet_DAIKIN_MasterStation_III_No_10.StartStopStatus_018.bPresVal AND
FB_BACnet_DAIKIN_MasterStation_III_No_10.StartStopStatus_019.bPresVal AND
FB_BACnet_DAIKIN_MasterStation_III_No_10.StartStopStatus_020.bPresVal AND
FB_BACnet_DAIKIN_MasterStation_III_No_10.StartStopStatus_021.bPresVal AND
FB_BACnet_DAIKIN_MasterStation_III_No_10.StartStopStatus_234.bPresVal
THEN
	nFloorStatus50 := 1;
ELSIF
NOT FB_BACnet_DAIKIN_MasterStation_III_No_10.StartStopStatus_000.bPresVal AND
NOT FB_BACnet_DAIKIN_MasterStation_III_No_10.StartStopStatus_001.bPresVal AND
NOT FB_BACnet_DAIKIN_MasterStation_III_No_10.StartStopStatus_002.bPresVal AND
NOT FB_BACnet_DAIKIN_MasterStation_III_No_10.StartStopStatus_003.bPresVal AND
NOT FB_BACnet_DAIKIN_MasterStation_III_No_10.StartStopStatus_004.bPresVal AND
NOT FB_BACnet_DAIKIN_MasterStation_III_No_10.StartStopStatus_005.bPresVal AND
NOT FB_BACnet_DAIKIN_MasterStation_III_No_10.StartStopStatus_006.bPresVal AND
NOT FB_BACnet_DAIKIN_MasterStation_III_No_10.StartStopStatus_007.bPresVal AND
NOT FB_BACnet_DAIKIN_MasterStation_III_No_10.StartStopStatus_008.bPresVal AND
NOT FB_BACnet_DAIKIN_MasterStation_III_No_10.StartStopStatus_009.bPresVal AND
NOT FB_BACnet_DAIKIN_MasterStation_III_No_10.StartStopStatus_010.bPresVal AND
NOT FB_BACnet_DAIKIN_MasterStation_III_No_10.StartStopStatus_011.bPresVal AND
NOT FB_BACnet_DAIKIN_MasterStation_III_No_10.StartStopStatus_012.bPresVal AND
NOT FB_BACnet_DAIKIN_MasterStation_III_No_10.StartStopStatus_013.bPresVal AND
NOT FB_BACnet_DAIKIN_MasterStation_III_No_10.StartStopStatus_014.bPresVal AND
NOT FB_BACnet_DAIKIN_MasterStation_III_No_10.StartStopStatus_015.bPresVal AND
NOT FB_BACnet_DAIKIN_MasterStation_III_No_10.StartStopStatus_016.bPresVal AND
NOT FB_BACnet_DAIKIN_MasterStation_III_No_10.StartStopStatus_017.bPresVal AND
NOT FB_BACnet_DAIKIN_MasterStation_III_No_10.StartStopStatus_018.bPresVal AND
NOT FB_BACnet_DAIKIN_MasterStation_III_No_10.StartStopStatus_019.bPresVal AND
NOT FB_BACnet_DAIKIN_MasterStation_III_No_10.StartStopStatus_020.bPresVal AND
NOT FB_BACnet_DAIKIN_MasterStation_III_No_10.StartStopStatus_021.bPresVal AND
NOT FB_BACnet_DAIKIN_MasterStation_III_No_10.StartStopStatus_234.bPresVal
THEN
	nFloorStatus50 := 0;
ELSE
	nFloorStatus50 := 2;
END_IF

//FloorStats 51
IF 
FB_BACnet_DAIKIN_MasterStation_III_No_10.StartStopStatus_064.bPresVal AND
FB_BACnet_DAIKIN_MasterStation_III_No_10.StartStopStatus_065.bPresVal AND
FB_BACnet_DAIKIN_MasterStation_III_No_10.StartStopStatus_066.bPresVal AND
FB_BACnet_DAIKIN_MasterStation_III_No_10.StartStopStatus_067.bPresVal AND
FB_BACnet_DAIKIN_MasterStation_III_No_10.StartStopStatus_068.bPresVal AND
FB_BACnet_DAIKIN_MasterStation_III_No_10.StartStopStatus_069.bPresVal AND
FB_BACnet_DAIKIN_MasterStation_III_No_10.StartStopStatus_070.bPresVal AND
FB_BACnet_DAIKIN_MasterStation_III_No_10.StartStopStatus_071.bPresVal AND
FB_BACnet_DAIKIN_MasterStation_III_No_10.StartStopStatus_072.bPresVal AND
FB_BACnet_DAIKIN_MasterStation_III_No_10.StartStopStatus_073.bPresVal AND
FB_BACnet_DAIKIN_MasterStation_III_No_10.StartStopStatus_074.bPresVal AND
FB_BACnet_DAIKIN_MasterStation_III_No_10.StartStopStatus_075.bPresVal AND
FB_BACnet_DAIKIN_MasterStation_III_No_10.StartStopStatus_076.bPresVal AND
FB_BACnet_DAIKIN_MasterStation_III_No_10.StartStopStatus_077.bPresVal AND
FB_BACnet_DAIKIN_MasterStation_III_No_10.StartStopStatus_078.bPresVal AND
FB_BACnet_DAIKIN_MasterStation_III_No_10.StartStopStatus_079.bPresVal AND
FB_BACnet_DAIKIN_MasterStation_III_No_10.StartStopStatus_080.bPresVal AND
FB_BACnet_DAIKIN_MasterStation_III_No_10.StartStopStatus_081.bPresVal AND
FB_BACnet_DAIKIN_MasterStation_III_No_10.StartStopStatus_082.bPresVal AND
FB_BACnet_DAIKIN_MasterStation_III_No_10.StartStopStatus_083.bPresVal AND
FB_BACnet_DAIKIN_MasterStation_III_No_10.StartStopStatus_084.bPresVal AND
FB_BACnet_DAIKIN_MasterStation_III_No_10.StartStopStatus_085.bPresVal AND
FB_BACnet_DAIKIN_MasterStation_III_No_10.StartStopStatus_235.bPresVal AND
FB_BACnet_DAIKIN_MasterStation_III_No_10.StartStopStatus_241.bPresVal AND
FB_BACnet_DAIKIN_MasterStation_III_No_10.StartStopStatus_112.bPresVal
THEN
	nFloorStatus51 := 1;
ELSIF
NOT FB_BACnet_DAIKIN_MasterStation_III_No_10.StartStopStatus_064.bPresVal AND
NOT FB_BACnet_DAIKIN_MasterStation_III_No_10.StartStopStatus_065.bPresVal AND
NOT FB_BACnet_DAIKIN_MasterStation_III_No_10.StartStopStatus_066.bPresVal AND
NOT FB_BACnet_DAIKIN_MasterStation_III_No_10.StartStopStatus_067.bPresVal AND
NOT FB_BACnet_DAIKIN_MasterStation_III_No_10.StartStopStatus_068.bPresVal AND
NOT FB_BACnet_DAIKIN_MasterStation_III_No_10.StartStopStatus_069.bPresVal AND
NOT FB_BACnet_DAIKIN_MasterStation_III_No_10.StartStopStatus_070.bPresVal AND
NOT FB_BACnet_DAIKIN_MasterStation_III_No_10.StartStopStatus_071.bPresVal AND
NOT FB_BACnet_DAIKIN_MasterStation_III_No_10.StartStopStatus_072.bPresVal AND
NOT FB_BACnet_DAIKIN_MasterStation_III_No_10.StartStopStatus_073.bPresVal AND
NOT FB_BACnet_DAIKIN_MasterStation_III_No_10.StartStopStatus_074.bPresVal AND
NOT FB_BACnet_DAIKIN_MasterStation_III_No_10.StartStopStatus_075.bPresVal AND
NOT FB_BACnet_DAIKIN_MasterStation_III_No_10.StartStopStatus_076.bPresVal AND
NOT FB_BACnet_DAIKIN_MasterStation_III_No_10.StartStopStatus_077.bPresVal AND
NOT FB_BACnet_DAIKIN_MasterStation_III_No_10.StartStopStatus_078.bPresVal AND
NOT FB_BACnet_DAIKIN_MasterStation_III_No_10.StartStopStatus_079.bPresVal AND
NOT FB_BACnet_DAIKIN_MasterStation_III_No_10.StartStopStatus_080.bPresVal AND
NOT FB_BACnet_DAIKIN_MasterStation_III_No_10.StartStopStatus_081.bPresVal AND
NOT FB_BACnet_DAIKIN_MasterStation_III_No_10.StartStopStatus_082.bPresVal AND
NOT FB_BACnet_DAIKIN_MasterStation_III_No_10.StartStopStatus_083.bPresVal AND
NOT FB_BACnet_DAIKIN_MasterStation_III_No_10.StartStopStatus_084.bPresVal AND
NOT FB_BACnet_DAIKIN_MasterStation_III_No_10.StartStopStatus_085.bPresVal AND
NOT FB_BACnet_DAIKIN_MasterStation_III_No_10.StartStopStatus_235.bPresVal AND
NOT FB_BACnet_DAIKIN_MasterStation_III_No_10.StartStopStatus_241.bPresVal AND
NOT FB_BACnet_DAIKIN_MasterStation_III_No_10.StartStopStatus_112.bPresVal
THEN
	nFloorStatus51 := 0;
ELSE
	nFloorStatus51 := 2;
END_IF

//FloorStats 52
IF 
FB_BACnet_DAIKIN_MasterStation_III_No_10.StartStopStatus_128.bPresVal AND
FB_BACnet_DAIKIN_MasterStation_III_No_10.StartStopStatus_129.bPresVal AND
FB_BACnet_DAIKIN_MasterStation_III_No_10.StartStopStatus_130.bPresVal AND
FB_BACnet_DAIKIN_MasterStation_III_No_10.StartStopStatus_131.bPresVal AND
FB_BACnet_DAIKIN_MasterStation_III_No_10.StartStopStatus_132.bPresVal AND
FB_BACnet_DAIKIN_MasterStation_III_No_10.StartStopStatus_133.bPresVal AND
FB_BACnet_DAIKIN_MasterStation_III_No_10.StartStopStatus_134.bPresVal AND
FB_BACnet_DAIKIN_MasterStation_III_No_10.StartStopStatus_135.bPresVal AND
FB_BACnet_DAIKIN_MasterStation_III_No_10.StartStopStatus_136.bPresVal AND
FB_BACnet_DAIKIN_MasterStation_III_No_10.StartStopStatus_137.bPresVal AND
FB_BACnet_DAIKIN_MasterStation_III_No_10.StartStopStatus_138.bPresVal AND
FB_BACnet_DAIKIN_MasterStation_III_No_10.StartStopStatus_139.bPresVal AND
FB_BACnet_DAIKIN_MasterStation_III_No_10.StartStopStatus_140.bPresVal AND
FB_BACnet_DAIKIN_MasterStation_III_No_10.StartStopStatus_141.bPresVal AND
FB_BACnet_DAIKIN_MasterStation_III_No_10.StartStopStatus_142.bPresVal AND
FB_BACnet_DAIKIN_MasterStation_III_No_10.StartStopStatus_143.bPresVal AND
FB_BACnet_DAIKIN_MasterStation_III_No_10.StartStopStatus_144.bPresVal AND
FB_BACnet_DAIKIN_MasterStation_III_No_10.StartStopStatus_145.bPresVal AND
FB_BACnet_DAIKIN_MasterStation_III_No_10.StartStopStatus_146.bPresVal AND
FB_BACnet_DAIKIN_MasterStation_III_No_10.StartStopStatus_147.bPresVal AND
FB_BACnet_DAIKIN_MasterStation_III_No_10.StartStopStatus_148.bPresVal AND
FB_BACnet_DAIKIN_MasterStation_III_No_10.StartStopStatus_149.bPresVal AND
FB_BACnet_DAIKIN_MasterStation_III_No_10.StartStopStatus_236.bPresVal
THEN
	nFloorStatus52 := 1;
ELSIF
NOT FB_BACnet_DAIKIN_MasterStation_III_No_10.StartStopStatus_128.bPresVal AND
NOT FB_BACnet_DAIKIN_MasterStation_III_No_10.StartStopStatus_129.bPresVal AND
NOT FB_BACnet_DAIKIN_MasterStation_III_No_10.StartStopStatus_130.bPresVal AND
NOT FB_BACnet_DAIKIN_MasterStation_III_No_10.StartStopStatus_131.bPresVal AND
NOT FB_BACnet_DAIKIN_MasterStation_III_No_10.StartStopStatus_132.bPresVal AND
NOT FB_BACnet_DAIKIN_MasterStation_III_No_10.StartStopStatus_133.bPresVal AND
NOT FB_BACnet_DAIKIN_MasterStation_III_No_10.StartStopStatus_134.bPresVal AND
NOT FB_BACnet_DAIKIN_MasterStation_III_No_10.StartStopStatus_135.bPresVal AND
NOT FB_BACnet_DAIKIN_MasterStation_III_No_10.StartStopStatus_136.bPresVal AND
NOT FB_BACnet_DAIKIN_MasterStation_III_No_10.StartStopStatus_137.bPresVal AND
NOT FB_BACnet_DAIKIN_MasterStation_III_No_10.StartStopStatus_138.bPresVal AND
NOT FB_BACnet_DAIKIN_MasterStation_III_No_10.StartStopStatus_139.bPresVal AND
NOT FB_BACnet_DAIKIN_MasterStation_III_No_10.StartStopStatus_140.bPresVal AND
NOT FB_BACnet_DAIKIN_MasterStation_III_No_10.StartStopStatus_141.bPresVal AND
NOT FB_BACnet_DAIKIN_MasterStation_III_No_10.StartStopStatus_142.bPresVal AND
NOT FB_BACnet_DAIKIN_MasterStation_III_No_10.StartStopStatus_143.bPresVal AND
NOT FB_BACnet_DAIKIN_MasterStation_III_No_10.StartStopStatus_144.bPresVal AND
NOT FB_BACnet_DAIKIN_MasterStation_III_No_10.StartStopStatus_145.bPresVal AND
NOT FB_BACnet_DAIKIN_MasterStation_III_No_10.StartStopStatus_146.bPresVal AND
NOT FB_BACnet_DAIKIN_MasterStation_III_No_10.StartStopStatus_147.bPresVal AND
NOT FB_BACnet_DAIKIN_MasterStation_III_No_10.StartStopStatus_148.bPresVal AND
NOT FB_BACnet_DAIKIN_MasterStation_III_No_10.StartStopStatus_149.bPresVal AND
NOT FB_BACnet_DAIKIN_MasterStation_III_No_10.StartStopStatus_236.bPresVal
THEN
	nFloorStatus52 := 0;
ELSE
	nFloorStatus52 := 2;
END_IF

//FloorStats 53
IF 
FB_BACnet_DAIKIN_MasterStation_III_No_10.StartStopStatus_192.bPresVal AND
FB_BACnet_DAIKIN_MasterStation_III_No_10.StartStopStatus_193.bPresVal AND
FB_BACnet_DAIKIN_MasterStation_III_No_10.StartStopStatus_194.bPresVal AND
FB_BACnet_DAIKIN_MasterStation_III_No_10.StartStopStatus_195.bPresVal AND
FB_BACnet_DAIKIN_MasterStation_III_No_10.StartStopStatus_196.bPresVal AND
FB_BACnet_DAIKIN_MasterStation_III_No_10.StartStopStatus_197.bPresVal AND
FB_BACnet_DAIKIN_MasterStation_III_No_10.StartStopStatus_198.bPresVal AND
FB_BACnet_DAIKIN_MasterStation_III_No_10.StartStopStatus_199.bPresVal AND
//FB_BACnet_DAIKIN_MasterStation_III_No_10.StartStopStatus_200.bPresVal AND
FB_BACnet_DAIKIN_MasterStation_III_No_10.StartStopStatus_201.bPresVal AND
FB_BACnet_DAIKIN_MasterStation_III_No_10.StartStopStatus_202.bPresVal AND
FB_BACnet_DAIKIN_MasterStation_III_No_10.StartStopStatus_203.bPresVal AND
FB_BACnet_DAIKIN_MasterStation_III_No_10.StartStopStatus_204.bPresVal AND
FB_BACnet_DAIKIN_MasterStation_III_No_10.StartStopStatus_205.bPresVal AND
FB_BACnet_DAIKIN_MasterStation_III_No_10.StartStopStatus_206.bPresVal AND
FB_BACnet_DAIKIN_MasterStation_III_No_10.StartStopStatus_207.bPresVal AND
FB_BACnet_DAIKIN_MasterStation_III_No_10.StartStopStatus_208.bPresVal AND
FB_BACnet_DAIKIN_MasterStation_III_No_10.StartStopStatus_209.bPresVal AND
FB_BACnet_DAIKIN_MasterStation_III_No_10.StartStopStatus_210.bPresVal AND
FB_BACnet_DAIKIN_MasterStation_III_No_10.StartStopStatus_211.bPresVal AND
FB_BACnet_DAIKIN_MasterStation_III_No_10.StartStopStatus_212.bPresVal AND
FB_BACnet_DAIKIN_MasterStation_III_No_10.StartStopStatus_213.bPresVal AND
FB_BACnet_DAIKIN_MasterStation_III_No_10.StartStopStatus_237.bPresVal AND
FB_BACnet_DAIKIN_MasterStation_III_No_10.StartStopStatus_243.bPresVal AND
FB_BACnet_DAIKIN_MasterStation_III_No_10.StartStopStatus_242.bPresVal
THEN
	nFloorStatus53 := 1;
ELSIF
NOT FB_BACnet_DAIKIN_MasterStation_III_No_10.StartStopStatus_192.bPresVal AND
NOT FB_BACnet_DAIKIN_MasterStation_III_No_10.StartStopStatus_193.bPresVal AND
NOT FB_BACnet_DAIKIN_MasterStation_III_No_10.StartStopStatus_194.bPresVal AND
NOT FB_BACnet_DAIKIN_MasterStation_III_No_10.StartStopStatus_195.bPresVal AND
NOT FB_BACnet_DAIKIN_MasterStation_III_No_10.StartStopStatus_196.bPresVal AND
NOT FB_BACnet_DAIKIN_MasterStation_III_No_10.StartStopStatus_197.bPresVal AND
NOT FB_BACnet_DAIKIN_MasterStation_III_No_10.StartStopStatus_198.bPresVal AND
NOT FB_BACnet_DAIKIN_MasterStation_III_No_10.StartStopStatus_199.bPresVal AND
//NOT FB_BACnet_DAIKIN_MasterStation_III_No_10.StartStopStatus_200.bPresVal AND
NOT FB_BACnet_DAIKIN_MasterStation_III_No_10.StartStopStatus_201.bPresVal AND
NOT FB_BACnet_DAIKIN_MasterStation_III_No_10.StartStopStatus_202.bPresVal AND
NOT FB_BACnet_DAIKIN_MasterStation_III_No_10.StartStopStatus_203.bPresVal AND
NOT FB_BACnet_DAIKIN_MasterStation_III_No_10.StartStopStatus_204.bPresVal AND
NOT FB_BACnet_DAIKIN_MasterStation_III_No_10.StartStopStatus_205.bPresVal AND
NOT FB_BACnet_DAIKIN_MasterStation_III_No_10.StartStopStatus_206.bPresVal AND
NOT FB_BACnet_DAIKIN_MasterStation_III_No_10.StartStopStatus_207.bPresVal AND
NOT FB_BACnet_DAIKIN_MasterStation_III_No_10.StartStopStatus_208.bPresVal AND
NOT FB_BACnet_DAIKIN_MasterStation_III_No_10.StartStopStatus_209.bPresVal AND
NOT FB_BACnet_DAIKIN_MasterStation_III_No_10.StartStopStatus_210.bPresVal AND
NOT FB_BACnet_DAIKIN_MasterStation_III_No_10.StartStopStatus_211.bPresVal AND
NOT FB_BACnet_DAIKIN_MasterStation_III_No_10.StartStopStatus_212.bPresVal AND
NOT FB_BACnet_DAIKIN_MasterStation_III_No_10.StartStopStatus_213.bPresVal AND
NOT FB_BACnet_DAIKIN_MasterStation_III_No_10.StartStopStatus_237.bPresVal AND
NOT FB_BACnet_DAIKIN_MasterStation_III_No_10.StartStopStatus_243.bPresVal AND
NOT FB_BACnet_DAIKIN_MasterStation_III_No_10.StartStopStatus_242.bPresVal
THEN
	nFloorStatus53 := 0;
ELSE
	nFloorStatus53 := 2;
END_IF

//FloorStats 55
IF 
FB_BACnet_DAIKIN_MasterStation_III_No_10.StartStopStatus_214.bPresVal AND
FB_BACnet_DAIKIN_MasterStation_III_No_10.StartStopStatus_215.bPresVal AND
FB_BACnet_DAIKIN_MasterStation_III_No_10.StartStopStatus_216.bPresVal AND
FB_BACnet_DAIKIN_MasterStation_III_No_10.StartStopStatus_217.bPresVal AND
FB_BACnet_DAIKIN_MasterStation_III_No_10.StartStopStatus_218.bPresVal AND
FB_BACnet_DAIKIN_MasterStation_III_No_10.StartStopStatus_219.bPresVal AND
FB_BACnet_DAIKIN_MasterStation_III_No_10.StartStopStatus_220.bPresVal AND
FB_BACnet_DAIKIN_MasterStation_III_No_10.StartStopStatus_221.bPresVal AND
FB_BACnet_DAIKIN_MasterStation_III_No_10.StartStopStatus_222.bPresVal AND
FB_BACnet_DAIKIN_MasterStation_III_No_10.StartStopStatus_223.bPresVal AND
FB_BACnet_DAIKIN_MasterStation_III_No_10.StartStopStatus_224.bPresVal AND
FB_BACnet_DAIKIN_MasterStation_III_No_10.StartStopStatus_225.bPresVal AND
FB_BACnet_DAIKIN_MasterStation_III_No_10.StartStopStatus_226.bPresVal AND
FB_BACnet_DAIKIN_MasterStation_III_No_10.StartStopStatus_227.bPresVal AND
FB_BACnet_DAIKIN_MasterStation_III_No_10.StartStopStatus_228.bPresVal AND
FB_BACnet_DAIKIN_MasterStation_III_No_10.StartStopStatus_229.bPresVal AND
FB_BACnet_DAIKIN_MasterStation_III_No_10.StartStopStatus_230.bPresVal AND
FB_BACnet_DAIKIN_MasterStation_III_No_10.StartStopStatus_231.bPresVal AND
FB_BACnet_DAIKIN_MasterStation_III_No_10.StartStopStatus_232.bPresVal AND
FB_BACnet_DAIKIN_MasterStation_III_No_10.StartStopStatus_233.bPresVal AND
FB_BACnet_DAIKIN_MasterStation_III_No_10.StartStopStatus_238.bPresVal
THEN
	nFloorStatus55 := 1;
ELSIF
NOT FB_BACnet_DAIKIN_MasterStation_III_No_10.StartStopStatus_214.bPresVal AND
NOT FB_BACnet_DAIKIN_MasterStation_III_No_10.StartStopStatus_215.bPresVal AND
NOT FB_BACnet_DAIKIN_MasterStation_III_No_10.StartStopStatus_216.bPresVal AND
NOT FB_BACnet_DAIKIN_MasterStation_III_No_10.StartStopStatus_217.bPresVal AND
NOT FB_BACnet_DAIKIN_MasterStation_III_No_10.StartStopStatus_218.bPresVal AND
NOT FB_BACnet_DAIKIN_MasterStation_III_No_10.StartStopStatus_219.bPresVal AND
NOT FB_BACnet_DAIKIN_MasterStation_III_No_10.StartStopStatus_220.bPresVal AND
NOT FB_BACnet_DAIKIN_MasterStation_III_No_10.StartStopStatus_221.bPresVal AND
NOT FB_BACnet_DAIKIN_MasterStation_III_No_10.StartStopStatus_222.bPresVal AND
NOT FB_BACnet_DAIKIN_MasterStation_III_No_10.StartStopStatus_223.bPresVal AND
NOT FB_BACnet_DAIKIN_MasterStation_III_No_10.StartStopStatus_224.bPresVal AND
NOT FB_BACnet_DAIKIN_MasterStation_III_No_10.StartStopStatus_225.bPresVal AND
NOT FB_BACnet_DAIKIN_MasterStation_III_No_10.StartStopStatus_226.bPresVal AND
NOT FB_BACnet_DAIKIN_MasterStation_III_No_10.StartStopStatus_227.bPresVal AND
NOT FB_BACnet_DAIKIN_MasterStation_III_No_10.StartStopStatus_228.bPresVal AND
NOT FB_BACnet_DAIKIN_MasterStation_III_No_10.StartStopStatus_229.bPresVal AND
NOT FB_BACnet_DAIKIN_MasterStation_III_No_10.StartStopStatus_230.bPresVal AND
NOT FB_BACnet_DAIKIN_MasterStation_III_No_10.StartStopStatus_231.bPresVal AND
NOT FB_BACnet_DAIKIN_MasterStation_III_No_10.StartStopStatus_232.bPresVal AND
NOT FB_BACnet_DAIKIN_MasterStation_III_No_10.StartStopStatus_233.bPresVal AND
NOT FB_BACnet_DAIKIN_MasterStation_III_No_10.StartStopStatus_238.bPresVal
THEN
	nFloorStatus55 := 0;
ELSE
	nFloorStatus55 := 2;
END_IF

//FloorStats PH1
IF 
FB_BACnet_DAIKIN_MasterStation_III_No_10.StartStopStatus_150.bPresVal AND
FB_BACnet_DAIKIN_MasterStation_III_No_10.StartStopStatus_151.bPresVal AND
FB_BACnet_DAIKIN_MasterStation_III_No_10.StartStopStatus_152.bPresVal AND
FB_BACnet_DAIKIN_MasterStation_III_No_10.StartStopStatus_153.bPresVal AND
FB_BACnet_DAIKIN_MasterStation_III_No_10.StartStopStatus_154.bPresVal AND
FB_BACnet_DAIKIN_MasterStation_III_No_10.StartStopStatus_155.bPresVal
THEN
	nFloorStatusPH1 := 1;
ELSIF
NOT FB_BACnet_DAIKIN_MasterStation_III_No_10.StartStopStatus_150.bPresVal AND
NOT FB_BACnet_DAIKIN_MasterStation_III_No_10.StartStopStatus_151.bPresVal AND
NOT FB_BACnet_DAIKIN_MasterStation_III_No_10.StartStopStatus_152.bPresVal AND
NOT FB_BACnet_DAIKIN_MasterStation_III_No_10.StartStopStatus_153.bPresVal AND
NOT FB_BACnet_DAIKIN_MasterStation_III_No_10.StartStopStatus_154.bPresVal AND
NOT FB_BACnet_DAIKIN_MasterStation_III_No_10.StartStopStatus_155.bPresVal
THEN
	nFloorStatusPH1 := 0;
ELSE
	nFloorStatusPH1 := 2;
END_IF

//FloorStats PH2
IF 
FB_BACnet_DAIKIN_MasterStation_III_No_10.StartStopStatus_156.bPresVal AND
FB_BACnet_DAIKIN_MasterStation_III_No_10.StartStopStatus_157.bPresVal AND
FB_BACnet_DAIKIN_MasterStation_III_No_10.StartStopStatus_158.bPresVal AND
FB_BACnet_DAIKIN_MasterStation_III_No_10.StartStopStatus_159.bPresVal AND
FB_BACnet_DAIKIN_MasterStation_III_No_10.StartStopStatus_160.bPresVal AND
FB_BACnet_DAIKIN_MasterStation_III_No_10.StartStopStatus_161.bPresVal AND
FB_BACnet_DAIKIN_MasterStation_III_No_10.StartStopStatus_162.bPresVal AND
FB_BACnet_DAIKIN_MasterStation_III_No_10.StartStopStatus_163.bPresVal AND
FB_BACnet_DAIKIN_MasterStation_III_No_10.StartStopStatus_164.bPresVal
THEN
	nFloorStatusPH2 := 1;
ELSIF
NOT FB_BACnet_DAIKIN_MasterStation_III_No_10.StartStopStatus_156.bPresVal AND
NOT FB_BACnet_DAIKIN_MasterStation_III_No_10.StartStopStatus_157.bPresVal AND
NOT FB_BACnet_DAIKIN_MasterStation_III_No_10.StartStopStatus_158.bPresVal AND
NOT FB_BACnet_DAIKIN_MasterStation_III_No_10.StartStopStatus_159.bPresVal AND
NOT FB_BACnet_DAIKIN_MasterStation_III_No_10.StartStopStatus_160.bPresVal AND
NOT FB_BACnet_DAIKIN_MasterStation_III_No_10.StartStopStatus_161.bPresVal AND
NOT FB_BACnet_DAIKIN_MasterStation_III_No_10.StartStopStatus_162.bPresVal AND
NOT FB_BACnet_DAIKIN_MasterStation_III_No_10.StartStopStatus_163.bPresVal AND
NOT FB_BACnet_DAIKIN_MasterStation_III_No_10.StartStopStatus_164.bPresVal
THEN
	nFloorStatusPH2 := 0;
ELSE
	nFloorStatusPH2 := 2;
END_IF

//FloorStats PH1
IF 
FB_BACnet_DAIKIN_MasterStation_III_No_10.StartStopStatus_165.bPresVal AND
FB_BACnet_DAIKIN_MasterStation_III_No_10.StartStopStatus_166.bPresVal AND
FB_BACnet_DAIKIN_MasterStation_III_No_10.StartStopStatus_167.bPresVal AND
FB_BACnet_DAIKIN_MasterStation_III_No_10.StartStopStatus_168.bPresVal AND
FB_BACnet_DAIKIN_MasterStation_III_No_10.StartStopStatus_169.bPresVal AND
FB_BACnet_DAIKIN_MasterStation_III_No_10.StartStopStatus_170.bPresVal AND
FB_BACnet_DAIKIN_MasterStation_III_No_10.StartStopStatus_171.bPresVal AND
FB_BACnet_DAIKIN_MasterStation_III_No_10.StartStopStatus_172.bPresVal AND
FB_BACnet_DAIKIN_MasterStation_III_No_10.StartStopStatus_173.bPresVal
THEN
	nFloorStatusPH3 := 1;
ELSIF
NOT FB_BACnet_DAIKIN_MasterStation_III_No_10.StartStopStatus_165.bPresVal AND
NOT FB_BACnet_DAIKIN_MasterStation_III_No_10.StartStopStatus_166.bPresVal AND
NOT FB_BACnet_DAIKIN_MasterStation_III_No_10.StartStopStatus_167.bPresVal AND
NOT FB_BACnet_DAIKIN_MasterStation_III_No_10.StartStopStatus_168.bPresVal AND
NOT FB_BACnet_DAIKIN_MasterStation_III_No_10.StartStopStatus_169.bPresVal AND
NOT FB_BACnet_DAIKIN_MasterStation_III_No_10.StartStopStatus_170.bPresVal AND
NOT FB_BACnet_DAIKIN_MasterStation_III_No_10.StartStopStatus_171.bPresVal AND
NOT FB_BACnet_DAIKIN_MasterStation_III_No_10.StartStopStatus_172.bPresVal AND
NOT FB_BACnet_DAIKIN_MasterStation_III_No_10.StartStopStatus_173.bPresVal
THEN
	nFloorStatusPH3 := 0;
ELSE
	nFloorStatusPH3 := 2;
END_IF

END_PROGRAM

